C05421=1105.460,240.179,428.078,179.305,14.265,151.128
C05422=1105.455,239.930,428.104,179.301,14.265,151.129
C05423=1105.449,239.682,428.131,179.297,14.266,151.129
C05424=1105.443,239.434,428.158,179.293,14.266,151.130
C05425=1105.437,239.185,428.184,179.289,14.266,151.131
C05426=1105.432,238.936,428.210,179.285,14.266,151.132
C05427=1105.426,238.688,428.237,179.281,14.266,151.133
C05428=1105.420,238.440,428.263,179.277,14.266,151.134
C05429=1105.415,238.191,428.289,179.274,14.266,151.135
C05430=1105.409,237.942,428.316,179.270,14.266,151.136
C05431=1105.404,237.693,428.342,179.266,14.266,151.137
C05432=1105.398,237.445,428.369,179.262,14.267,151.138
C05433=1105.393,237.197,428.395,179.258,14.267,151.139
C05434=1105.387,236.948,428.421,179.254,14.267,151.139
C05435=1105.379,236.586,428.459,179.248,14.266,151.141
C05436=1105.370,236.224,428.498,179.242,14.267,151.142
C05437=1105.363,235.862,428.536,179.237,14.267,151.143
C05438=1105.354,235.500,428.574,179.231,14.268,151.145
C05439=1105.348,235.252,428.600,179.227,14.268,151.146
C05440=1105.342,235.003,428.626,179.223,14.268,151.147
C05441=1105.336,234.754,428.653,179.220,14.268,151.147
C05442=1105.331,234.506,428.678,179.216,14.268,151.148
C05443=1105.326,234.257,428.704,179.211,14.268,151.149
C05444=1105.320,234.009,428.731,179.208,14.268,151.150
C05445=1105.315,233.760,428.757,179.204,14.268,151.151
C05446=1105.308,233.512,428.783,179.200,14.268,151.152
C05447=1105.303,233.263,428.809,179.196,14.269,151.153
C05448=1105.297,233.014,428.835,179.192,14.269,151.154
C05449=1105.292,232.765,428.861,179.188,14.269,151.155
C05450=1105.286,232.516,428.887,179.184,14.269,151.156
C05451=1105.280,232.269,428.913,179.180,14.269,151.157
C05452=1105.275,232.020,428.939,179.176,14.269,151.157
C05453=1105.269,231.771,428.965,179.172,14.270,151.159
C05454=1105.264,231.522,428.991,179.168,14.270,151.159
C05455=1105.257,231.274,429.017,179.164,14.270,151.160
C05456=1105.252,231.025,429.043,179.160,14.270,151.161
C05457=1105.247,230.777,429.068,179.156,14.270,151.162
C05458=1105.241,230.529,429.095,179.152,14.270,151.163
C05459=1105.235,230.280,429.120,179.148,14.270,151.164
C05460=1105.229,230.031,429.146,179.145,14.271,151.165
C05461=1105.224,229.782,429.172,179.141,14.271,151.166
C05462=1105.218,229.533,429.198,179.137,14.272,151.167
C05463=1105.213,229.286,429.224,179.133,14.272,151.168
C05464=1105.206,229.037,429.249,179.129,14.272,151.169
C05465=1105.201,228.788,429.275,179.125,14.272,151.170
C05466=1105.195,228.539,429.301,179.121,14.272,151.171
C05467=1105.189,228.290,429.326,179.117,14.272,151.171
C05468=1105.184,228.041,429.352,179.113,14.272,151.172
C05469=1105.178,227.794,429.378,179.109,14.273,151.173
C05470=1105.172,227.545,429.404,179.105,14.273,151.174
C05471=1105.167,227.296,429.430,179.101,14.273,151.175
C05472=1105.161,227.047,429.455,179.097,14.273,151.176
C05473=1105.156,226.799,429.481,179.094,14.274,151.177
C05474=1105.150,226.550,429.506,179.090,14.274,151.178
C05475=1105.144,226.301,429.532,179.086,14.274,151.179
C05476=1105.138,226.053,429.557,179.082,14.275,151.180
C05477=1105.133,225.804,429.583,179.078,14.275,151.181
C05478=1105.127,225.556,429.608,179.074,14.275,151.182
C05479=1105.121,225.307,429.634,179.070,14.275,151.183
C05480=1105.115,225.058,429.660,179.066,14.276,151.184
C05481=1105.110,224.810,429.685,179.062,14.276,151.185
C05482=1105.104,224.561,429.710,179.058,14.276,151.185
C05483=1105.099,224.312,429.736,179.055,14.276,151.186
C05484=1105.092,224.064,429.762,179.051,14.277,151.187
C05485=1105.088,223.815,429.787,179.047,14.277,151.188
C05486=1105.081,223.567,429.813,179.043,14.277,151.189
C05487=1105.074,223.196,429.851,179.037,14.277,151.191
C05488=1105.065,222.825,429.888,179.031,14.278,151.192
C05489=1105.057,222.456,429.926,179.026,14.278,151.193
C05490=1105.048,222.085,429.964,179.020,14.279,151.195
C05491=1105.042,221.836,429.990,179.016,14.279,151.196
C05492=1105.037,221.588,430.014,179.012,14.279,151.197
C05493=1105.031,221.339,430.040,179.008,14.280,151.198
C05494=1105.025,221.090,430.065,179.004,14.280,151.199
C05495=1105.020,220.842,430.090,179.000,14.280,151.199
C05496=1105.014,220.593,430.116,178.996,14.280,151.201
C05497=1105.008,220.344,430.141,178.992,14.280,151.201
C05498=1105.003,220.096,430.166,178.989,14.281,151.202
C05499=1104.997,219.847,430.191,178.985,14.282,151.203
C05500=1104.991,219.597,430.217,178.981,14.282,151.204
C05501=1104.986,219.349,430.241,178.977,14.282,151.205
C05502=1104.980,219.101,430.267,178.973,14.282,151.206
C05503=1104.973,218.852,430.292,178.969,14.282,151.207
C05504=1104.969,218.603,430.317,178.965,14.283,151.208
C05505=1104.963,218.355,430.342,178.961,14.283,151.209
C05506=1104.957,218.107,430.367,178.957,14.284,151.210
C05507=1104.951,217.857,430.392,178.954,14.284,151.211
C05508=1104.946,217.608,430.418,178.949,14.284,151.212
C05509=1104.940,217.360,430.442,178.945,14.284,151.213
C05510=1104.934,217.111,430.467,178.942,14.285,151.214
C05511=1104.929,216.863,430.492,178.937,14.285,151.215
C05512=1104.923,216.614,430.517,178.933,14.285,151.216
C05513=1104.918,216.366,430.543,178.930,14.286,151.216
C05514=1104.912,216.116,430.567,178.926,14.286,151.218
C05515=1104.906,215.868,430.593,178.922,14.287,151.218
C05516=1104.900,215.619,430.617,178.918,14.287,151.219
C05517=1104.894,215.370,430.642,178.914,14.287,151.220
C05518=1104.890,215.121,430.667,178.910,14.287,151.221
C05519=1104.883,214.873,430.692,178.906,14.287,151.222
C05520=1104.878,214.624,430.717,178.903,14.288,151.223
C05521=1104.872,214.375,430.742,178.899,14.289,151.224
C05522=1104.867,214.127,430.766,178.895,14.289,151.225
C05523=1104.860,213.878,430.792,178.891,14.289,151.226
C05524=1104.856,213.629,430.816,178.887,14.289,151.227
C05525=1104.850,213.380,430.841,178.883,14.289,151.228
C05526=1104.844,213.132,430.866,178.879,14.291,151.229
C05527=1104.839,212.883,430.891,178.876,14.291,151.230
C05528=1104.833,212.635,430.916,178.871,14.291,151.231
C05529=1104.827,212.386,430.940,178.867,14.291,151.232
C05530=1104.822,212.137,430.964,178.864,14.291,151.233
C05531=1104.816,211.888,430.990,178.859,14.292,151.234
C05532=1104.810,211.640,431.014,178.856,14.293,151.235
C05533=1104.804,211.390,431.039,178.852,14.293,151.236
C05534=1104.799,211.142,431.064,178.848,14.293,151.237
C05535=1104.793,210.893,431.088,178.844,14.293,151.237
C05536=1104.787,210.645,431.113,178.840,14.294,151.238
C05537=1104.782,210.396,431.137,178.836,14.294,151.239
C05538=1104.776,210.147,431.162,178.833,14.295,151.240
C05539=1104.768,209.781,431.198,178.826,14.295,151.242
C05540=1104.759,209.413,431.234,178.821,14.296,151.243
C05541=1104.752,209.046,431.270,178.815,14.296,151.245
C05542=1104.743,208.679,431.307,178.810,14.297,151.246
C05543=1104.720,207.682,431.405,178.783,14.296,151.252
C05544=1104.714,207.433,431.429,178.779,14.297,151.253
C05545=1104.709,207.184,431.453,178.774,14.298,151.254
C05546=1104.703,206.936,431.477,178.770,14.299,151.256
C05547=1104.697,206.687,431.502,178.766,14.301,151.257
C05548=1104.691,206.438,431.526,178.761,14.302,151.258
C05549=1104.686,206.190,431.550,178.758,14.303,151.259
C05550=1104.679,205.941,431.574,178.753,14.304,151.260
C05551=1104.674,205.692,431.599,178.749,14.306,151.262
C05552=1104.668,205.443,431.623,178.745,14.307,151.263
C05553=1104.663,205.194,431.647,178.741,14.308,151.264
C05554=1104.657,204.946,431.671,178.737,14.309,151.265
C05555=1104.651,204.697,431.696,178.733,14.311,151.266
C05556=1104.646,204.448,431.720,178.728,14.312,151.268
C05557=1104.640,204.200,431.744,178.724,14.312,151.269
C05558=1104.634,203.951,431.768,178.720,14.314,151.270
C05559=1104.628,203.702,431.793,178.716,14.315,151.271
C05560=1104.623,203.453,431.817,178.712,14.316,151.272
C05561=1104.617,203.205,431.840,178.708,14.317,151.273
C05562=1104.611,202.956,431.865,178.704,14.319,151.275
C05563=1104.606,202.707,431.889,178.699,14.319,151.276
C05564=1104.600,202.458,431.912,178.695,14.321,151.277
C05565=1104.594,202.209,431.937,178.691,14.322,151.278
C05566=1104.588,201.961,431.961,178.687,14.323,151.279
C05567=1104.583,201.712,431.985,178.683,14.324,151.281
C05568=1104.577,201.463,432.009,178.678,14.325,151.282
C05569=1104.571,201.215,432.033,178.674,14.327,151.283
C05570=1104.566,200.965,432.057,178.670,14.327,151.284
C05571=1104.559,200.716,432.081,178.666,14.329,151.285
C05572=1104.554,200.468,432.105,178.662,14.330,151.287
C05573=1104.548,200.220,432.129,178.658,14.331,151.288
C05574=1104.542,199.970,432.153,178.654,14.332,151.289
C05575=1104.536,199.721,432.176,178.650,14.334,151.290
C05576=1104.531,199.473,432.200,178.645,14.335,151.291
C05577=1104.525,199.225,432.224,178.642,14.336,151.292
C05578=1104.520,198.975,432.248,178.637,14.337,151.294
C05579=1104.513,198.726,432.272,178.633,14.339,151.295
C05580=1104.508,198.478,432.296,178.629,14.339,151.296
C05581=1104.502,198.229,432.320,178.625,14.341,151.297
C05582=1104.496,197.980,432.343,178.621,14.342,151.298
C05583=1104.491,197.731,432.367,178.617,14.343,151.299
C05584=1104.485,197.482,432.390,178.613,14.344,151.301
C05585=1104.479,197.234,432.414,178.609,14.345,151.302
C05586=1104.473,196.985,432.438,178.605,14.347,151.303
C05587=1104.468,196.736,432.462,178.600,14.348,151.304
C05588=1104.462,196.487,432.486,178.597,14.349,151.305
C05589=1104.457,196.238,432.509,178.592,14.350,151.307
C05590=1104.451,195.990,432.533,178.589,14.351,151.308
C05591=1104.444,195.741,432.557,178.584,14.352,151.309
C05592=1104.439,195.492,432.580,178.581,14.353,151.310
C05593=1104.433,195.243,432.604,178.576,14.354,151.311
C05594=1104.428,194.994,432.627,178.572,14.356,151.312
C05595=1104.422,194.746,432.651,178.568,14.356,151.313
C05596=1104.416,194.497,432.674,178.564,14.358,151.315
C05597=1104.410,194.248,432.699,178.560,14.359,151.316
C05598=1104.405,193.999,432.722,178.555,14.360,151.317
C05599=1104.399,193.751,432.745,178.552,14.361,151.318
C05600=1104.394,193.501,432.769,178.547,14.362,151.319
C05601=1104.388,193.252,432.792,178.544,14.363,151.320
C05602=1104.382,193.004,432.815,178.540,14.364,151.321
C05603=1104.377,192.755,432.839,178.536,14.365,151.323
C05604=1104.370,192.483,432.865,178.531,14.366,151.324
C05605=1104.364,192.212,432.890,178.527,14.367,151.325
C05606=1104.358,191.941,432.916,178.523,14.369,151.326
C05607=1104.352,191.670,432.941,178.518,14.370,151.328
C05608=1104.346,191.421,432.964,178.514,14.371,151.329
C05609=1104.341,191.172,432.989,178.510,14.372,151.330
C05610=1104.335,190.923,433.012,178.506,14.373,151.331
C05611=1104.329,190.674,433.034,178.502,14.375,151.332
C05612=1104.323,190.425,433.059,178.498,14.375,151.333
C05613=1104.318,190.176,433.082,178.494,14.377,151.334
C05614=1104.312,189.927,433.105,178.490,14.378,151.336
C05615=1104.306,189.678,433.128,178.486,14.379,151.337
C05616=1104.301,189.430,433.152,178.482,14.379,151.338
C05617=1104.295,189.181,433.175,178.478,14.380,151.339
C05618=1104.290,188.932,433.198,178.474,14.382,151.340
C05619=1104.284,188.683,433.221,178.470,14.382,151.341
C05620=1104.278,188.435,433.245,178.466,14.384,151.342
C05621=1104.273,188.186,433.268,178.462,14.385,151.343
C05622=1104.267,187.937,433.291,178.458,14.386,151.345
C05623=1104.261,187.688,433.314,178.454,14.386,151.346
C05624=1104.256,187.439,433.338,178.450,14.388,151.347
C05625=1104.251,187.190,433.361,178.446,14.389,151.348
C05626=1104.245,186.941,433.384,178.442,14.390,151.349
C05627=1104.239,186.693,433.407,178.438,14.391,151.350
C05628=1104.233,186.444,433.430,178.434,14.392,151.351
C05629=1104.228,186.195,433.454,178.430,14.393,151.352
C05630=1104.222,185.946,433.477,178.426,14.393,151.353
C05631=1104.217,185.697,433.499,178.422,14.395,151.354
C05632=1104.211,185.449,433.522,178.418,14.396,151.356
C05633=1104.206,185.200,433.545,178.414,14.397,151.357
C05634=1104.200,184.951,433.568,178.410,14.398,151.358
C05635=1104.194,184.702,433.591,178.407,14.399,151.359
C05636=1104.189,184.453,433.614,178.402,14.400,151.360
C05637=1104.183,184.204,433.637,178.399,14.401,151.361
C05638=1104.176,183.954,433.660,178.394,14.402,151.362
C05639=1104.171,183.706,433.683,178.391,14.403,151.364
C05640=1104.165,183.457,433.706,178.386,14.404,151.365
C05641=1104.159,183.208,433.729,178.383,14.405,151.366
C05642=1104.154,182.959,433.752,178.378,14.406,151.367
C05643=1104.148,182.710,433.775,178.375,14.408,151.368
C05644=1104.141,182.461,433.797,178.371,14.408,151.369
C05645=1104.136,182.212,433.820,178.367,14.410,151.370
C05646=1104.130,181.964,433.843,178.363,14.411,151.371
C05647=1104.125,181.715,433.866,178.359,14.412,151.372
C05648=1104.119,181.466,433.889,178.355,14.412,151.374
C05649=1104.113,181.218,433.912,178.351,14.414,151.375
C05650=1104.108,180.969,433.935,178.347,14.415,151.376
C05651=1104.101,180.720,433.957,178.343,14.416,151.377
C05652=1104.096,180.471,433.979,178.339,14.417,151.378
C05653=1104.090,180.222,434.002,178.336,14.418,151.379
C05654=1104.084,179.973,434.025,178.331,14.419,151.380
C05655=1104.078,179.724,434.048,178.328,14.420,151.381
C05656=1104.073,179.475,434.071,178.323,14.421,151.382
C05657=1104.067,179.226,434.093,178.320,14.422,151.383
C05658=1104.061,178.977,434.116,178.316,14.423,151.385
C05659=1104.055,178.728,434.139,178.312,14.424,151.386
C05660=1104.049,178.479,434.161,178.308,14.425,151.387
C05661=1104.044,178.231,434.184,178.304,14.426,151.388
C05662=1104.038,177.982,434.206,178.300,14.427,151.389
C05663=1104.032,177.733,434.229,178.297,14.428,151.390
C05664=1104.027,177.484,434.252,178.292,14.429,151.391
C05665=1104.021,177.234,434.274,178.288,14.430,151.392
C05666=1104.015,176.985,434.297,178.284,14.431,151.393
C05667=1104.009,176.737,434.319,178.280,14.432,151.394
C05668=1104.003,176.465,434.344,178.277,14.433,151.395
C05669=1103.997,176.194,434.368,178.272,14.434,151.397
C05670=1103.991,175.922,434.393,178.268,14.435,151.398
C05671=1103.985,175.650,434.418,178.263,14.436,151.399
C05672=1103.979,175.401,434.439,178.260,14.437,151.400
C05673=1103.973,175.152,434.462,178.255,14.438,151.401
C05674=1103.967,174.903,434.485,178.252,14.439,151.402
C05675=1103.961,174.654,434.507,178.248,14.439,151.403
C05676=1103.956,174.406,434.529,178.244,14.441,151.404
C05677=1103.951,174.156,434.552,178.240,14.441,151.405
C05678=1103.945,173.907,434.575,178.237,14.443,151.407
C05679=1103.939,173.658,434.596,178.232,14.443,151.408
C05680=1103.934,173.410,434.619,178.229,14.445,151.409
C05681=1103.928,173.160,434.641,178.225,14.445,151.410
C05682=1103.922,172.912,434.663,178.221,14.447,151.411
C05683=1103.916,172.662,434.686,178.217,14.447,151.412
C05684=1103.911,172.414,434.708,178.214,14.448,151.413
C05685=1103.905,172.165,434.730,178.209,14.449,151.414
C05686=1103.899,171.916,434.753,178.206,14.450,151.415
C05687=1103.894,171.667,434.775,178.202,14.451,151.416
C05688=1103.888,171.419,434.797,178.198,14.452,151.417
C05689=1103.883,171.169,434.819,178.194,14.453,151.418
C05690=1103.877,170.920,434.842,178.191,14.453,151.419
C05691=1103.871,170.671,434.864,178.187,14.454,151.420
C05692=1103.866,170.422,434.886,178.183,14.455,151.421
C05693=1103.859,170.174,434.908,178.179,14.456,151.422
C05694=1103.854,169.924,434.930,178.175,14.457,151.423
C05695=1103.849,169.675,434.952,178.172,14.458,151.424
C05696=1103.843,169.427,434.974,178.168,14.459,151.425
C05697=1103.837,169.177,434.997,178.164,14.459,151.426
C05698=1103.832,168.929,435.018,178.160,14.461,151.427
C05699=1103.826,168.680,435.041,178.156,14.461,151.428
C05700=1103.821,168.430,435.063,178.153,14.462,151.429
C05701=1103.815,168.182,435.084,178.149,14.463,151.431
C05702=1103.809,167.933,435.107,178.145,14.464,151.432
C05703=1103.803,167.684,435.129,178.141,14.464,151.432
C05704=1103.798,167.435,435.151,178.138,14.466,151.434
C05705=1103.792,167.186,435.172,178.134,14.466,151.435
C05706=1103.786,166.937,435.195,178.130,14.467,151.436
C05707=1103.782,166.688,435.217,178.126,14.468,151.437
C05708=1103.775,166.439,435.239,178.123,14.469,151.438
C05709=1103.771,166.190,435.261,178.119,14.470,151.439
C05710=1103.764,165.941,435.282,178.115,14.470,151.440
C05711=1103.759,165.692,435.305,178.111,14.471,151.441
C05712=1103.753,165.443,435.327,178.107,14.472,151.442
C05713=1103.748,165.194,435.349,178.104,14.473,151.443
C05714=1103.742,164.945,435.370,178.100,14.473,151.444
C05715=1103.737,164.696,435.392,178.096,14.475,151.445
C05716=1103.731,164.447,435.414,178.092,14.475,151.446
C05717=1103.726,164.198,435.436,178.089,14.476,151.447
C05718=1103.719,163.949,435.458,178.085,14.477,151.448
C05719=1103.714,163.700,435.480,178.081,14.478,151.449
C05720=1103.708,163.451,435.502,178.077,14.478,151.450
C05721=1103.703,163.202,435.524,178.074,14.479,151.451
C05722=1103.697,162.953,435.545,178.070,14.480,151.452
C05723=1103.692,162.704,435.567,178.067,14.481,151.453
C05724=1103.686,162.455,435.589,178.062,14.481,151.454
C05725=1103.681,162.207,435.610,178.059,14.482,151.455
C05726=1103.675,161.957,435.632,178.055,14.483,151.456
C05727=1103.670,161.709,435.653,178.052,14.484,151.457
C05728=1103.664,161.459,435.676,178.048,14.485,151.458
C05729=1103.659,161.211,435.697,178.045,14.485,151.459
C05730=1103.653,160.961,435.719,178.040,14.486,151.460
C05731=1103.647,160.713,435.740,178.037,14.487,151.461
C05732=1103.641,160.440,435.764,178.033,14.488,151.462
C05733=1103.634,160.168,435.788,178.028,14.489,151.463
C05734=1103.628,159.896,435.811,178.025,14.490,151.464
C05735=1103.622,159.624,435.835,178.021,14.491,151.465
C05736=1103.617,159.375,435.856,178.017,14.491,151.466
C05737=1103.610,159.126,435.878,178.013,14.492,151.467
C05738=1103.605,158.877,435.899,178.009,14.493,151.468
C05739=1103.599,158.628,435.921,178.006,14.494,151.469
C05740=1103.594,158.379,435.942,178.002,14.494,151.470
C05741=1103.588,158.130,435.963,177.998,14.495,151.471
C05742=1103.582,157.881,435.985,177.995,14.496,151.472
C05743=1103.576,157.632,436.006,177.991,14.497,151.473
C05744=1103.571,157.383,436.028,177.987,14.497,151.474
C05745=1103.565,157.134,436.050,177.984,14.498,151.475
C05746=1103.560,156.885,436.070,177.980,14.499,151.476
C05747=1103.554,156.635,436.092,177.977,14.500,151.477
C05748=1103.548,156.387,436.113,177.972,14.500,151.478
C05749=1103.542,156.138,436.135,177.969,14.501,151.479
C05750=1103.538,155.888,436.156,177.965,14.502,151.480
C05751=1103.531,155.639,436.178,177.962,14.503,151.481
C05752=1103.526,155.391,436.199,177.958,14.503,151.482
C05753=1103.520,155.142,436.220,177.955,14.504,151.483
C05754=1103.515,154.892,436.241,177.950,14.505,151.484
C05755=1103.509,154.644,436.262,177.947,14.506,151.485
C05756=1103.503,154.395,436.284,177.943,14.506,151.485
C05757=1103.498,154.145,436.305,177.940,14.507,151.487
C05758=1103.491,153.896,436.326,177.936,14.508,151.487
C05759=1103.486,153.648,436.347,177.933,14.508,151.488
C05760=1103.480,153.398,436.368,177.929,14.509,151.489
C05761=1103.474,153.149,436.390,177.925,14.510,151.490
C05762=1103.469,152.901,436.411,177.922,14.510,151.491
C05763=1103.463,152.651,436.432,177.918,14.512,151.492
C05764=1103.457,152.403,436.453,177.914,14.512,151.493
C05765=1103.451,152.153,436.475,177.911,14.513,151.494
C05766=1103.447,151.904,436.496,177.907,14.513,151.495
C05767=1103.441,151.655,436.517,177.904,14.514,151.496
C05768=1103.435,151.406,436.538,177.900,14.515,151.497
C05769=1103.430,151.157,436.559,177.897,14.516,151.498
C05770=1103.423,150.908,436.580,177.893,14.516,151.499
C05771=1103.418,150.659,436.601,177.889,14.517,151.500
C05772=1103.412,150.410,436.621,177.886,14.518,151.501
C05773=1103.406,150.161,436.643,177.882,14.518,151.502
C05774=1103.401,149.912,436.664,177.879,14.519,151.503
C05775=1103.395,149.663,436.685,177.875,14.519,151.504
C05776=1103.390,149.413,436.706,177.872,14.521,151.505
C05777=1103.384,149.165,436.727,177.868,14.521,151.506
C05778=1103.379,148.916,436.748,177.864,14.522,151.506
C05779=1103.373,148.666,436.769,177.861,14.522,151.507
C05780=1103.367,148.417,436.790,177.857,14.523,151.508
C05781=1103.362,148.169,436.811,177.853,14.523,151.509
C05782=1103.356,147.919,436.832,177.850,14.524,151.510
C05783=1103.350,147.670,436.852,177.846,14.525,151.511
C05784=1103.344,147.422,436.873,177.843,14.526,151.512
C05785=1103.338,147.172,436.894,177.839,14.526,151.513
C05786=1103.333,146.923,436.915,177.836,14.527,151.514
C05787=1103.328,146.674,436.936,177.832,14.527,151.515
C05788=1103.322,146.424,436.957,177.829,14.528,151.516
C05789=1103.315,146.176,436.978,177.825,14.529,151.517
C05790=1103.310,145.927,436.998,177.822,14.530,151.518
C05791=1103.304,145.677,437.019,177.817,14.530,151.519
C05792=1103.299,145.429,437.040,177.814,14.531,151.520
C05793=1103.293,145.180,437.060,177.810,14.531,151.520
C05794=1103.287,144.930,437.081,177.807,14.532,151.521
C05795=1103.281,144.682,437.103,177.803,14.533,151.522
C05796=1103.275,144.409,437.125,177.800,14.534,151.523
C05797=1103.269,144.136,437.148,177.796,14.534,151.524
C05798=1103.264,143.864,437.170,177.792,14.535,151.525
C05799=1103.257,143.592,437.192,177.788,14.535,151.526
C05800=1103.251,143.342,437.213,177.785,14.536,151.527
C05801=1103.245,143.094,437.234,177.781,14.537,151.528
C05802=1103.240,142.845,437.255,177.778,14.537,151.529
C05803=1103.234,142.596,437.275,177.774,14.538,151.530
C05804=1103.228,142.346,437.296,177.770,14.539,151.531
C05805=1103.223,142.097,437.316,177.768,14.539,151.532
C05806=1103.217,141.848,437.337,177.764,14.539,151.532
C05807=1103.211,141.600,437.357,177.761,14.540,151.533
C05808=1103.206,141.351,437.378,177.757,14.541,151.534
C05809=1103.200,141.101,437.399,177.754,14.541,151.535
C05810=1103.194,140.852,437.419,177.750,14.542,151.536
C05811=1103.189,140.603,437.439,177.746,14.543,151.537
C05812=1103.184,140.354,437.460,177.743,14.543,151.538
C05813=1103.178,140.105,437.480,177.739,14.544,151.539
C05814=1103.172,139.855,437.501,177.735,14.544,151.540
C05815=1103.166,139.606,437.521,177.733,14.545,151.541
C05816=1103.160,139.358,437.542,177.729,14.545,151.541
C05817=1103.155,139.109,437.563,177.726,14.546,151.542
C05818=1103.149,138.860,437.583,177.722,14.546,151.543
C05819=1103.144,138.611,437.603,177.719,14.547,151.544
C05820=1103.137,138.361,437.623,177.715,14.547,151.545
C05821=1103.132,138.112,437.644,177.711,14.548,151.546
C05822=1103.127,137.863,437.665,177.708,14.548,151.547
C05823=1103.121,137.614,437.685,177.705,14.549,151.548
C05824=1103.116,137.365,437.705,177.702,14.550,151.549
C05825=1103.110,137.116,437.725,177.698,14.550,151.549
C05826=1103.104,136.866,437.745,177.694,14.551,151.550
C05827=1103.098,136.617,437.765,177.691,14.551,151.551
C05828=1103.093,136.368,437.786,177.688,14.552,151.552
C05829=1103.087,136.119,437.806,177.684,14.552,151.553
C05830=1103.081,135.870,437.826,177.681,14.553,151.554
C05831=1103.075,135.621,437.846,177.677,14.553,151.555
C05832=1103.070,135.372,437.867,177.674,14.554,151.556
C05833=1103.064,135.122,437.887,177.670,14.554,151.556
C05834=1103.058,134.873,437.908,177.667,14.555,151.557
C05835=1103.052,134.624,437.928,177.663,14.555,151.558
C05836=1103.047,134.375,437.947,177.660,14.556,151.559
C05837=1103.041,134.126,437.967,177.656,14.556,151.560
C05838=1103.035,133.877,437.987,177.653,14.557,151.561
C05839=1103.030,133.628,438.008,177.649,14.557,151.562
C05840=1103.024,133.379,438.028,177.646,14.558,151.562
C05841=1103.019,133.129,438.048,177.643,14.558,151.563
C05842=1103.013,132.881,438.068,177.640,14.559,151.564
C05843=1103.008,132.631,438.088,177.636,14.560,151.565
C05844=1103.002,132.383,438.108,177.633,14.560,151.566
C05845=1102.996,132.134,438.128,177.630,14.561,151.567
C05846=1102.990,131.883,438.148,177.626,14.561,151.568
C05847=1102.984,131.635,438.168,177.623,14.561,151.568
C05848=1102.978,131.386,438.188,177.619,14.562,151.569
C05849=1102.973,131.137,438.209,177.616,14.563,151.570
C05850=1102.968,130.887,438.228,177.612,14.562,151.571
C05851=1102.962,130.638,438.248,177.609,14.563,151.572
C05852=1102.956,130.390,438.268,177.605,14.564,151.573
C05853=1102.951,130.140,438.288,177.602,14.564,151.574
C05854=1102.945,129.891,438.308,177.598,14.565,151.574
C05855=1102.939,129.642,438.328,177.596,14.565,151.575
C05856=1102.933,129.393,438.347,177.592,14.566,151.576
C05857=1102.928,129.144,438.368,177.589,14.566,151.577
C05858=1102.921,128.894,438.388,177.586,14.567,151.578
C05859=1102.915,128.645,438.407,177.582,14.567,151.579
C05860=1102.909,128.373,438.429,177.578,14.567,151.580
C05861=1102.903,128.100,438.451,177.575,14.568,151.580
C05862=1102.897,127.827,438.472,177.571,14.569,151.581
C05863=1102.890,127.555,438.494,177.567,14.569,151.582
C05864=1102.885,127.306,438.513,177.564,14.569,151.583
C05865=1102.880,127.057,438.533,177.560,14.570,151.584
C05866=1102.874,126.807,438.553,177.557,14.570,151.585
C05867=1102.868,126.558,438.573,177.554,14.571,151.586
C05868=1102.862,126.310,438.593,177.551,14.571,151.586
C05869=1102.856,126.060,438.612,177.548,14.572,151.587
C05870=1102.850,125.811,438.632,177.544,14.572,151.588
C05871=1102.845,125.562,438.652,177.541,14.572,151.589
C05872=1102.839,125.313,438.672,177.537,14.573,151.590
C05873=1102.834,125.063,438.691,177.534,14.573,151.590
C05874=1102.828,124.814,438.710,177.530,14.574,151.591
C05875=1102.822,124.565,438.730,177.527,14.574,151.592
C05876=1102.816,124.316,438.749,177.524,14.574,151.593
C05877=1102.810,124.067,438.769,177.521,14.575,151.594
C05878=1102.805,123.817,438.789,177.518,14.575,151.595
C05879=1102.799,123.568,438.809,177.514,14.575,151.595
C05880=1102.794,123.319,438.828,177.511,14.576,151.596
C05881=1102.788,123.070,438.847,177.508,14.576,151.597
C05882=1102.782,122.821,438.867,177.504,14.577,151.598
C05883=1102.777,122.572,438.886,177.501,14.577,151.599
C05884=1102.771,122.323,438.906,177.498,14.577,151.599
C05885=1102.765,122.074,438.926,177.494,14.577,151.600
C05886=1102.759,121.824,438.945,177.491,14.578,151.601
C05887=1102.754,121.575,438.965,177.488,14.578,151.602
C05888=1102.748,121.326,438.985,177.485,14.579,151.603
C05889=1102.743,121.076,439.004,177.481,14.579,151.603
C05890=1102.738,120.828,439.023,177.478,14.580,151.604
C05891=1102.732,120.579,439.043,177.475,14.580,151.605
C05892=1102.726,120.329,439.062,177.472,14.580,151.606
C05893=1102.720,120.080,439.081,177.469,14.581,151.607
C05894=1102.715,119.830,439.100,177.465,14.581,151.607
C05895=1102.709,119.582,439.120,177.462,14.581,151.608
C05896=1102.704,119.333,439.139,177.459,14.581,151.609
C05897=1102.698,119.083,439.158,177.456,14.582,151.610
C05898=1102.692,118.834,439.178,177.452,14.582,151.611
C05899=1102.686,118.585,439.197,177.449,14.582,151.611
C05900=1102.680,118.336,439.217,177.445,14.582,151.612
C05901=1102.675,118.086,439.236,177.443,14.583,151.613
C05902=1102.670,117.838,439.255,177.440,14.583,151.613
C05903=1102.664,117.588,439.274,177.436,14.583,151.614
C05904=1102.658,117.339,439.294,177.433,14.584,151.615
C05905=1102.653,117.089,439.313,177.430,14.584,151.616
C05906=1102.648,116.841,439.332,177.427,14.585,151.617
C05907=1102.642,116.592,439.352,177.423,14.585,151.617
C05908=1102.636,116.342,439.371,177.420,14.585,151.618
C05909=1102.630,116.093,439.390,177.416,14.585,151.619
C05910=1102.625,115.844,439.409,177.414,14.585,151.620
C05911=1102.619,115.595,439.428,177.410,14.585,151.620
C05912=1102.614,115.345,439.447,177.407,14.586,151.621
C05913=1102.608,115.096,439.467,177.404,14.586,151.622
C05914=1102.603,114.847,439.486,177.401,14.586,151.623
C05915=1102.597,114.598,439.505,177.398,14.587,151.623
C05916=1102.592,114.348,439.524,177.394,14.587,151.624
C05917=1102.586,114.099,439.543,177.392,14.587,151.625
C05918=1102.580,113.850,439.562,177.388,14.587,151.626
C05919=1102.574,113.601,439.581,177.385,14.588,151.626
C05920=1102.569,113.352,439.600,177.382,14.588,151.627
C05921=1102.563,113.102,439.619,177.379,14.588,151.628
C05922=1102.558,112.853,439.638,177.376,14.589,151.629
C05923=1102.551,112.604,439.657,177.372,14.588,151.629
C05924=1102.545,112.331,439.678,177.368,14.589,151.630
C05925=1102.539,112.059,439.699,177.366,14.589,151.631
C05926=1102.533,111.786,439.719,177.362,14.589,151.632
C05927=1102.527,111.513,439.741,177.358,14.590,151.633
C05928=1102.521,111.265,439.759,177.355,14.590,151.634
C05929=1102.515,111.016,439.778,177.352,14.591,151.634
C05930=1102.510,110.766,439.797,177.349,14.590,151.635
C05931=1102.504,110.517,439.816,177.346,14.591,151.636
C05932=1102.498,110.268,439.834,177.342,14.591,151.637
C05933=1102.493,110.018,439.853,177.340,14.591,151.637
C05934=1102.487,109.769,439.873,177.336,14.591,151.638
C05935=1102.481,109.520,439.891,177.333,14.592,151.639
C05936=1102.475,109.271,439.910,177.330,14.592,151.640
C05937=1102.470,109.021,439.929,177.327,14.592,151.640
C05938=1102.464,108.772,439.947,177.324,14.592,151.641
C05939=1102.459,108.523,439.966,177.321,14.592,151.642
C05940=1102.453,108.274,439.986,177.318,14.593,151.642
C05941=1102.446,108.024,440.004,177.314,14.593,151.643
C05942=1102.441,107.776,440.023,177.311,14.593,151.644
C05943=1102.435,107.526,440.041,177.308,14.593,151.645
C05944=1102.430,107.277,440.060,177.305,14.594,151.645
C05945=1102.424,107.028,440.079,177.302,14.594,151.646
C05946=1102.418,106.779,440.098,177.299,14.594,151.647
C05947=1102.413,106.529,440.116,177.296,14.594,151.647
C05948=1102.408,106.280,440.135,177.292,14.594,151.648
C05949=1102.401,106.031,440.154,177.290,14.595,151.649
C05950=1102.396,105.781,440.172,177.286,14.594,151.650
C05951=1102.390,105.532,440.191,177.283,14.595,151.650
C05952=1102.384,105.283,440.210,177.281,14.595,151.651
C05953=1102.379,105.034,440.228,177.277,14.595,151.652
C05954=1102.373,104.784,440.247,177.274,14.596,151.653
C05955=1102.368,104.536,440.266,177.271,14.595,151.653
C05956=1102.362,104.286,440.283,177.268,14.596,151.654
C05957=1102.356,104.036,440.303,177.264,14.595,151.655
C05958=1102.350,103.788,440.321,177.262,14.596,151.655
C05959=1102.345,103.538,440.340,177.259,14.596,151.656
C05960=1102.339,103.290,440.358,177.256,14.596,151.657
C05961=1102.334,103.040,440.376,177.253,14.597,151.657
C05962=1102.328,102.790,440.396,177.249,14.596,151.658
C05963=1102.322,102.542,440.414,177.247,14.596,151.659
C05964=1102.317,102.292,440.432,177.243,14.596,151.660
C05965=1102.311,102.043,440.451,177.241,14.596,151.660
C05966=1102.306,101.793,440.469,177.238,14.597,151.661
C05967=1102.300,101.545,440.487,177.234,14.597,151.662
C05968=1102.294,101.295,440.506,177.232,14.597,151.662
C05969=1102.289,101.046,440.524,177.228,14.597,151.663
C05970=1102.283,100.796,440.543,177.225,14.597,151.664
C05971=1102.277,100.547,440.561,177.222,14.597,151.664
C05972=1102.271,100.298,440.579,177.219,14.597,151.665
C05973=1102.266,100.049,440.598,177.216,14.598,151.666
C05974=1102.260,99.800,440.616,177.213,14.597,151.666
C05975=1102.254,99.550,440.634,177.210,14.598,151.667
C05976=1102.249,99.301,440.653,177.207,14.598,151.668
C05977=1102.243,99.051,440.671,177.204,14.598,151.668
C05978=1102.238,98.803,440.689,177.200,14.598,151.669
C05979=1102.232,98.553,440.707,177.198,14.598,151.670
C05980=1102.225,98.304,440.726,177.195,14.599,151.671
C05981=1102.220,98.054,440.744,177.191,14.598,151.671
C05982=1102.214,97.805,440.763,177.189,14.599,151.672
C05983=1102.208,97.556,440.780,177.185,14.598,151.673
C05984=1102.203,97.306,440.799,177.183,14.599,151.673
C05985=1102.197,97.058,440.817,177.180,14.599,151.674
C05986=1102.191,96.808,440.835,177.176,14.599,151.675
C05987=1102.186,96.559,440.853,177.174,14.599,151.675
C05988=1102.180,96.286,440.873,177.170,14.599,151.676
C05989=1102.173,96.014,440.893,177.167,14.599,151.677
C05990=1102.167,95.742,440.913,177.164,14.599,151.678
C05991=1102.161,95.469,440.933,177.161,14.599,151.678
C05992=1102.156,95.220,440.951,177.158,14.600,151.679
C05993=1102.150,94.970,440.969,177.155,14.599,151.680
C05994=1102.144,94.722,440.987,177.152,14.600,151.680
C05995=1102.138,94.472,441.005,177.149,14.600,151.681
C05996=1102.133,94.223,441.023,177.146,14.600,151.682
C05997=1102.127,93.973,441.041,177.143,14.600,151.682
C05998=1102.122,93.723,441.059,177.139,14.600,151.683
C05999=1102.115,93.474,441.078,177.137,14.600,151.684
C06000=1102.110,93.225,441.095,177.134,14.599,151.684
C06001=1102.104,92.976,441.113,177.131,14.600,151.685
C06002=1102.099,92.726,441.131,177.128,14.600,151.685
C06003=1102.094,92.477,441.149,177.125,14.600,151.686
C06004=1102.087,92.228,441.168,177.122,14.600,151.687
C06005=1102.082,91.979,441.185,177.119,14.599,151.687
C06006=1102.076,91.730,441.203,177.116,14.600,151.688
C06007=1102.071,91.480,441.221,177.114,14.600,151.689
C06008=1102.065,91.231,441.239,177.110,14.599,151.689
C06009=1102.060,90.982,441.256,177.108,14.600,151.690
C06010=1102.054,90.732,441.274,177.104,14.599,151.691
C06011=1102.048,90.484,441.293,177.102,14.599,151.691
C06012=1102.042,90.234,441.311,177.099,14.600,151.692
C06013=1102.036,89.985,441.328,177.096,14.599,151.693
C06014=1102.031,89.735,441.347,177.093,14.600,151.693
C06015=1102.025,89.486,441.364,177.090,14.600,151.694
C06016=1102.020,89.237,441.382,177.087,14.600,151.695
C06017=1102.014,88.987,441.400,177.084,14.600,151.695
C06018=1102.008,88.738,441.417,177.081,14.600,151.696
C06019=1102.002,88.488,441.435,177.078,14.600,151.696
C06020=1101.996,88.239,441.453,177.075,14.600,151.697
C06021=1101.991,87.990,441.470,177.072,14.600,151.698
C06022=1101.985,87.740,441.488,177.070,14.600,151.698
C06023=1101.979,87.491,441.506,177.066,14.600,151.699
C06024=1101.974,87.242,441.523,177.064,14.600,151.700
C06025=1101.968,86.993,441.541,177.060,14.599,151.700
C06026=1101.962,86.744,441.559,177.058,14.599,151.701
C06027=1101.957,86.495,441.577,177.055,14.600,151.702
C06028=1101.950,86.245,441.594,177.052,14.600,151.702
C06029=1101.945,85.996,441.612,177.049,14.600,151.703
C06030=1101.939,85.747,441.630,177.046,14.599,151.703
C06031=1101.933,85.497,441.648,177.044,14.599,151.704
C06032=1101.928,85.248,441.665,177.041,14.600,151.705
C06033=1101.922,84.999,441.683,177.037,14.599,151.705
C06034=1101.916,84.749,441.700,177.035,14.599,151.706
C06035=1101.911,84.500,441.717,177.032,14.599,151.707
C06036=1101.905,84.250,441.735,177.029,14.599,151.707
C06037=1101.899,84.001,441.753,177.026,14.599,151.708
C06038=1101.894,83.752,441.770,177.023,14.599,151.708
C06039=1101.888,83.503,441.788,177.021,14.599,151.709
C06040=1101.883,83.254,441.806,177.018,14.599,151.710
C06041=1101.877,83.003,441.823,177.015,14.599,151.710
C06042=1101.871,82.754,441.840,177.012,14.599,151.711
C06043=1101.866,82.505,441.858,177.009,14.598,151.711
C06044=1101.860,82.256,441.875,177.006,14.598,151.712
C06045=1101.853,82.007,441.893,177.004,14.599,151.713
C06046=1101.848,81.757,441.910,177.000,14.598,151.713
C06047=1101.843,81.508,441.927,176.998,14.598,151.714
C06048=1101.837,81.259,441.945,176.995,14.598,151.715
C06049=1101.831,81.009,441.963,176.992,14.598,151.715
C06050=1101.826,80.760,441.980,176.990,14.598,151.716
C06051=1101.820,80.511,441.997,176.986,14.598,151.716
C06052=1101.814,80.238,442.017,176.984,14.598,151.717
C06053=1101.808,79.966,442.035,176.980,14.598,151.718
C06054=1101.801,79.693,442.054,176.977,14.597,151.718
C06055=1101.796,79.421,442.073,176.974,14.597,151.719
C06056=1101.790,79.171,442.091,176.971,14.597,151.719
C06057=1101.785,78.921,442.108,176.969,14.597,151.720
C06058=1101.778,78.673,442.125,176.966,14.597,151.721
C06059=1101.773,78.424,442.142,176.963,14.596,151.721
C06060=1101.767,78.173,442.160,176.960,14.597,151.722
C06061=1101.761,77.924,442.177,176.958,14.597,151.722
C06062=1101.756,77.675,442.195,176.955,14.596,151.723
C06063=1101.750,77.426,442.211,176.952,14.596,151.724
C06064=1101.744,77.177,442.228,176.949,14.596,151.724
C06065=1101.738,76.927,442.246,176.946,14.596,151.725
C06066=1101.733,76.677,442.263,176.944,14.596,151.725
C06067=1101.727,76.429,442.280,176.940,14.595,151.726
C06068=1101.722,76.179,442.297,176.938,14.596,151.726
C06069=1101.716,75.930,442.315,176.935,14.596,151.727
C06070=1101.710,75.681,442.331,176.932,14.595,151.728
C06071=1101.704,75.431,442.349,176.930,14.595,151.728
C06072=1101.699,75.181,442.366,176.926,14.595,151.729
C06073=1101.693,74.933,442.383,176.924,14.595,151.729
C06074=1101.687,74.684,442.400,176.921,14.595,151.730
C06075=1101.682,74.434,442.417,176.918,14.595,151.731
C06076=1101.676,74.185,442.435,176.916,14.595,151.731
C06077=1101.670,73.935,442.451,176.913,14.594,151.732
C06078=1101.664,73.686,442.469,176.910,14.594,151.732
C06079=1101.659,73.436,442.486,176.908,14.594,151.733
C06080=1101.653,73.187,442.502,176.904,14.593,151.733
C06081=1101.648,72.938,442.520,176.902,14.593,151.734
C06082=1101.642,72.688,442.536,176.899,14.594,151.735
C06083=1101.636,72.439,442.553,176.896,14.593,151.735
C06084=1101.631,72.190,442.570,176.894,14.593,151.736
C06085=1101.624,71.940,442.588,176.891,14.593,151.736
C06086=1101.619,71.691,442.604,176.888,14.592,151.737
C06087=1101.614,71.441,442.621,176.886,14.592,151.737
C06088=1101.607,71.192,442.638,176.883,14.593,151.738
C06089=1101.602,70.943,442.655,176.880,14.592,151.739
C06090=1101.596,70.694,442.672,176.878,14.592,151.739
C06091=1101.591,70.444,442.689,176.874,14.591,151.740
C06092=1101.585,70.194,442.706,176.872,14.591,151.740
C06093=1101.579,69.946,442.723,176.869,14.591,151.741
C06094=1101.574,69.696,442.740,176.866,14.591,151.741
C06095=1101.568,69.447,442.756,176.864,14.591,151.742
C06096=1101.562,69.197,442.774,176.861,14.591,151.742
C06097=1101.556,68.948,442.790,176.858,14.590,151.743
C06098=1101.551,68.698,442.807,176.855,14.590,151.743
C06099=1101.544,68.449,442.824,176.853,14.590,151.744
C06100=1101.539,68.200,442.841,176.850,14.590,151.745
C06101=1101.533,67.950,442.857,176.848,14.590,151.745
C06102=1101.528,67.701,442.874,176.844,14.589,151.746
C06103=1101.522,67.452,442.891,176.842,14.589,151.746
C06104=1101.517,67.202,442.908,176.840,14.589,151.747
C06105=1101.511,66.953,442.924,176.836,14.588,151.747
C06106=1101.505,66.703,442.941,176.834,14.588,151.748
C06107=1101.499,66.454,442.958,176.832,14.588,151.748
C06108=1101.494,66.205,442.975,176.828,14.588,151.749
C06109=1101.488,65.955,442.991,176.826,14.588,151.749
C06110=1101.482,65.706,443.007,176.824,14.587,151.750
C06111=1101.477,65.456,443.024,176.820,14.587,151.751
C06112=1101.471,65.208,443.041,176.818,14.587,151.751
C06113=1101.465,64.958,443.058,176.816,14.587,151.752
C06114=1101.459,64.709,443.074,176.812,14.586,151.752
C06115=1101.454,64.459,443.091,176.810,14.586,151.753
C06116=1101.447,64.186,443.109,176.807,14.585,151.753
C06117=1101.441,63.914,443.127,176.804,14.586,151.754
C06118=1101.434,63.641,443.145,176.801,14.585,151.754
C06119=1101.428,63.368,443.163,176.799,14.585,151.755
C06120=1101.422,63.120,443.180,176.795,14.585,151.756
C06121=1101.417,62.870,443.196,176.793,14.585,151.756
C06122=1101.411,62.621,443.213,176.791,14.584,151.757
C06123=1101.405,62.371,443.229,176.787,14.584,151.757
C06124=1101.399,62.122,443.245,176.785,14.584,151.758
C06125=1101.394,61.872,443.262,176.783,14.584,151.758
C06126=1101.388,61.623,443.278,176.779,14.583,151.759
C06127=1101.382,61.374,443.295,176.777,14.583,151.759
C06128=1101.376,61.124,443.311,176.775,14.583,151.760
C06129=1101.370,60.875,443.327,176.771,14.583,151.760
C06130=1101.365,60.625,443.344,176.769,14.582,151.761
C06131=1101.359,60.376,443.360,176.767,14.582,151.761
C06132=1101.353,60.127,443.376,176.763,14.582,151.762
C06133=1101.347,59.877,443.393,176.761,14.581,151.762
C06134=1101.342,59.628,443.410,176.759,14.582,151.763
C06135=1101.336,59.378,443.426,176.756,14.581,151.763
C06136=1101.330,59.129,443.442,176.753,14.581,151.764
C06137=1101.324,58.880,443.458,176.751,14.580,151.764
C06138=1101.318,58.630,443.475,176.748,14.580,151.765
C06139=1101.313,58.381,443.491,176.746,14.580,151.765
C06140=1101.307,58.131,443.508,176.743,14.580,151.766
C06141=1101.301,57.882,443.524,176.740,14.579,151.766
C06142=1101.295,57.633,443.540,176.738,14.579,151.767
C06143=1101.289,57.383,443.556,176.735,14.579,151.767
C06144=1101.284,57.135,443.572,176.732,14.578,151.768
C06145=1101.278,56.885,443.589,176.730,14.578,151.768
C06146=1101.273,56.635,443.605,176.727,14.578,151.769
C06147=1101.267,56.386,443.621,176.724,14.577,151.769
C06148=1101.261,56.136,443.637,176.722,14.577,151.770
C06149=1101.255,55.887,443.654,176.720,14.577,151.770
C06150=1101.249,55.637,443.670,176.717,14.577,151.771
C06151=1101.243,55.388,443.686,176.714,14.576,151.772
C06152=1101.238,55.138,443.702,176.712,14.576,151.772
C06153=1101.232,54.889,443.718,176.710,14.576,151.773
C06154=1101.227,54.640,443.734,176.706,14.575,151.773
C06155=1101.221,54.391,443.751,176.704,14.575,151.774
C06156=1101.215,54.141,443.767,176.702,14.575,151.774
C06157=1101.209,53.891,443.782,176.699,14.574,151.775
C06158=1101.203,53.642,443.799,176.696,14.574,151.775
C06159=1101.197,53.393,443.815,176.694,14.574,151.776
C06160=1101.192,53.144,443.831,176.691,14.573,151.776
C06161=1101.187,52.894,443.847,176.689,14.573,151.776
C06162=1101.181,52.644,443.863,176.686,14.573,151.777
C06163=1101.175,52.395,443.879,176.683,14.572,151.777
C06164=1101.169,52.146,443.896,176.681,14.571,151.778
C06165=1101.164,51.896,443.911,176.679,14.572,151.778
C06166=1101.158,51.647,443.927,176.676,14.571,151.779
C06167=1101.152,51.398,443.943,176.673,14.570,151.779
C06168=1101.147,51.148,443.959,176.671,14.570,151.780
C06169=1101.141,50.898,443.975,176.668,14.569,151.780
C06170=1101.135,50.649,443.991,176.666,14.569,151.781
C06171=1101.130,50.400,444.007,176.663,14.569,151.781
C06172=1101.124,50.150,444.023,176.661,14.569,151.782
C06173=1101.118,49.901,444.039,176.658,14.568,151.782
C06174=1101.112,49.651,444.055,176.656,14.568,151.783
C06175=1101.107,49.402,444.071,176.653,14.568,151.783
C06176=1101.101,49.153,444.087,176.650,14.567,151.784
C06177=1101.095,48.903,444.102,176.648,14.567,151.784
C06178=1101.089,48.654,444.119,176.646,14.566,151.784
C06179=1101.084,48.404,444.134,176.643,14.566,151.785
C06180=1101.078,48.131,444.151,176.641,14.565,151.786
C06181=1101.072,47.859,444.169,176.637,14.565,151.786
C06182=1101.066,47.586,444.187,176.635,14.565,151.787
C06183=1101.060,47.313,444.204,176.632,14.564,151.787
C06184=1101.054,47.063,444.219,176.630,14.564,151.788
C06185=1101.048,46.814,444.236,176.628,14.563,151.788
C06186=1101.043,46.565,444.251,176.625,14.562,151.788
C06187=1101.037,46.315,444.267,176.622,14.562,151.789
C06188=1101.031,46.065,444.283,176.620,14.562,151.789
C06189=1101.026,45.816,444.299,176.617,14.561,151.790
C06190=1101.020,45.567,444.314,176.615,14.561,151.790
C06191=1101.015,45.317,444.330,176.613,14.561,151.791
C06192=1101.009,45.067,444.346,176.610,14.560,151.791
C06193=1101.004,44.819,444.362,176.607,14.559,151.792
C06194=1100.998,44.569,444.377,176.605,14.559,151.792
C06195=1100.992,44.319,444.393,176.603,14.559,151.792
C06196=1100.987,44.070,444.409,176.600,14.558,151.793
C06197=1100.981,43.820,444.424,176.598,14.558,151.793
C06198=1100.975,43.571,444.440,176.595,14.558,151.794
C06199=1100.970,43.322,444.455,176.593,14.557,151.794
C06200=1100.964,43.073,444.471,176.590,14.556,151.795
C06201=1100.958,42.823,444.487,176.588,14.556,151.795
C06202=1100.953,42.573,444.502,176.586,14.556,151.796
C06203=1100.946,42.324,444.518,176.583,14.555,151.796
C06204=1100.941,42.074,444.533,176.580,14.555,151.797
C06205=1100.935,41.826,444.549,176.578,14.555,151.797
C06206=1100.930,41.576,444.565,176.576,14.554,151.797
C06207=1100.924,41.326,444.580,176.573,14.553,151.798
C06208=1100.918,41.077,444.595,176.571,14.553,151.798
C06209=1100.912,40.827,444.611,176.569,14.553,151.799
C06210=1100.907,40.578,444.627,176.566,14.552,151.799
C06211=1100.901,40.329,444.642,176.563,14.551,151.800
C06212=1100.895,40.079,444.657,176.561,14.551,151.800
C06213=1100.889,39.829,444.673,176.559,14.551,151.801
C06214=1100.884,39.580,444.688,176.556,14.550,151.801
C06215=1100.878,39.331,444.704,176.554,14.550,151.801
C06216=1100.872,39.081,444.719,176.551,14.550,151.802
C06217=1100.867,38.832,444.734,176.548,14.549,151.802
C06218=1100.861,38.582,444.750,176.546,14.548,151.803
C06219=1100.856,38.333,444.766,176.544,14.548,151.803
C06220=1100.849,38.083,444.781,176.542,14.548,151.804
C06221=1100.844,37.833,444.796,176.539,14.547,151.804
C06222=1100.839,37.584,444.812,176.537,14.546,151.804
C06223=1100.832,37.335,444.827,176.535,14.546,151.805
C06224=1100.827,37.086,444.842,176.532,14.546,151.805
C06225=1100.821,36.836,444.857,176.529,14.545,151.806
C06226=1100.815,36.586,444.873,176.527,14.545,151.806
C06227=1100.810,36.337,444.888,176.525,14.544,151.807
C06228=1100.803,36.088,444.904,176.522,14.543,151.807
C06229=1100.798,35.838,444.919,176.520,14.543,151.807
C06230=1100.792,35.589,444.934,176.518,14.543,151.808
C06231=1100.786,35.339,444.949,176.515,14.542,151.808
C06232=1100.781,35.090,444.965,176.513,14.541,151.809
C06233=1100.775,34.840,444.980,176.510,14.541,151.809
C06234=1100.769,34.590,444.995,176.508,14.541,151.810
C06235=1100.763,34.342,445.010,176.506,14.540,151.810
C06236=1100.757,34.092,445.026,176.503,14.540,151.810
C06237=1100.751,33.843,445.040,176.501,14.539,151.811
C06238=1100.746,33.593,445.056,176.499,14.539,151.811
C06239=1100.740,33.343,445.072,176.496,14.539,151.812
C06240=1100.734,33.094,445.086,176.493,14.538,151.812
C06241=1100.729,32.844,445.102,176.491,14.537,151.813
C06242=1100.723,32.595,445.116,176.489,14.537,151.813
C06243=1100.717,32.345,445.132,176.487,14.537,151.813
C06244=1100.711,32.073,445.148,176.484,14.536,151.814
C06245=1100.704,31.800,445.164,176.482,14.535,151.814
C06246=1100.698,31.527,445.182,176.478,14.535,151.815
C06247=1100.692,31.254,445.198,176.476,14.535,151.815
C06248=1100.686,31.005,445.213,176.474,14.534,151.816
C06249=1100.680,30.755,445.228,176.471,14.533,151.816
C06250=1100.676,30.506,445.243,176.469,14.533,151.816
C06251=1100.669,30.256,445.258,176.467,14.532,151.817
C06252=1100.664,30.007,445.273,176.465,14.532,151.817
C06253=1100.658,29.757,445.288,176.462,14.531,151.818
C06254=1100.652,29.508,445.302,176.460,14.531,151.818
C06255=1100.646,29.258,445.318,176.458,14.530,151.819
C06256=1100.641,29.009,445.333,176.455,14.530,151.819
C06257=1100.635,28.759,445.348,176.452,14.529,151.819
C06258=1100.629,28.510,445.363,176.451,14.528,151.820
C06259=1100.624,28.260,445.378,176.448,14.528,151.820
C06260=1100.618,28.011,445.393,176.446,14.528,151.821
C06261=1100.611,27.762,445.408,176.443,14.527,151.821
C06262=1100.606,27.512,445.423,176.441,14.526,151.821
C06263=1100.600,27.263,445.438,176.439,14.526,151.822
C06264=1100.595,27.013,445.452,176.437,14.526,151.822
C06265=1100.589,26.763,445.467,176.434,14.526,151.823
C06266=1100.583,26.514,445.482,176.432,14.524,151.823
C06267=1100.577,26.264,445.497,176.430,14.524,151.823
C06268=1100.572,26.015,445.512,176.427,14.524,151.824
C06269=1100.565,25.766,445.527,176.425,14.523,151.824
C06270=1100.560,25.516,445.542,176.422,14.522,151.825
C06271=1100.555,25.267,445.556,176.420,14.522,151.825
C06272=1100.548,25.017,445.571,176.418,14.521,151.825
C06273=1100.543,24.768,445.586,176.416,14.521,151.826
C06274=1100.537,24.518,445.601,176.413,14.520,151.826
C06275=1100.531,24.269,445.616,176.411,14.520,151.827
C06276=1100.526,24.019,445.630,176.409,14.519,151.827
C06277=1100.520,23.770,445.645,176.406,14.519,151.827
C06278=1100.514,23.520,445.660,176.405,14.518,151.828
C06279=1100.508,23.271,445.675,176.402,14.517,151.828
C06280=1100.503,23.021,445.689,176.399,14.517,151.829
C06281=1100.497,22.772,445.704,176.397,14.517,151.829
C06282=1100.491,22.523,445.719,176.395,14.516,151.829
C06283=1100.485,22.273,445.734,176.393,14.516,151.830
C06284=1100.480,22.023,445.748,176.390,14.515,151.830
C06285=1100.473,21.773,445.763,176.388,14.514,151.831
C06286=1100.468,21.524,445.777,176.386,14.514,151.831
C06287=1100.463,21.275,445.792,176.384,14.513,151.831
C06288=1100.457,21.025,445.807,176.381,14.512,151.832
C06289=1100.451,20.776,445.821,176.379,14.512,151.832
C06290=1100.445,20.526,445.835,176.377,14.511,151.832
C06291=1100.440,20.276,445.851,176.375,14.511,151.833
C06292=1100.434,20.027,445.865,176.373,14.511,151.833
C06293=1100.428,19.777,445.880,176.370,14.510,151.834
C06294=1100.422,19.528,445.894,176.368,14.509,151.834
C06295=1100.416,19.279,445.909,176.366,14.509,151.834
C06296=1100.410,19.029,445.923,176.363,14.508,151.835
C06297=1100.405,18.780,445.938,176.361,14.508,151.835
C06298=1100.399,18.529,445.952,176.359,14.507,151.835
C06299=1100.393,18.280,445.967,176.356,14.506,151.836
C06300=1100.387,18.032,445.982,176.354,14.506,151.836
C06301=1100.381,17.781,445.996,176.352,14.506,151.837
C06302=1100.376,17.532,446.010,176.350,14.505,151.837
C06303=1100.370,17.283,446.024,176.347,14.504,151.837
C06304=1100.364,17.033,446.040,176.345,14.504,151.838
C06305=1100.359,16.783,446.054,176.343,14.503,151.838
C06306=1100.353,16.534,446.068,176.341,14.503,151.838
C06307=1100.347,16.284,446.083,176.339,14.502,151.839
C06308=1100.341,16.013,446.098,176.336,14.501,151.839
C06309=1100.335,15.742,446.114,176.334,14.500,151.840
C06310=1100.328,15.470,446.130,176.331,14.500,151.840
C06311=1100.322,15.199,446.145,176.329,14.499,151.841
C06312=1100.317,14.949,446.160,176.326,14.499,151.841
C06313=1100.311,14.700,446.175,176.325,14.498,151.841
C06314=1100.305,14.450,446.188,176.322,14.498,151.842
C06315=1100.299,14.201,446.203,176.319,14.497,151.842
C06316=1100.293,13.951,446.217,176.318,14.496,151.842
C06317=1100.288,13.702,446.232,176.315,14.496,151.843
C06318=1100.282,13.452,446.246,176.313,14.496,151.843
C06319=1100.276,13.202,446.260,176.311,14.495,151.843
C06320=1100.270,12.954,446.274,176.308,14.494,151.844
C06321=1100.263,12.703,446.288,176.306,14.494,151.844
C06322=1100.258,12.454,446.303,176.304,14.493,151.845
C06323=1100.252,12.205,446.317,176.302,14.492,151.845
C06324=1100.246,11.955,446.331,176.300,14.492,151.845
C06325=1100.240,11.706,446.345,176.298,14.491,151.846
C06326=1100.235,11.456,446.359,176.295,14.490,151.846
C06327=1100.229,11.206,446.374,176.293,14.490,151.847
C06328=1100.223,10.957,446.388,176.291,14.489,151.847
C06329=1100.218,10.707,446.402,176.289,14.489,151.847
C06330=1100.212,10.458,446.416,176.287,14.489,151.848
C06331=1100.206,10.208,446.431,176.285,14.488,151.848
C06332=1100.199,9.959,446.444,176.282,14.487,151.848
C06333=1100.194,9.710,446.459,176.280,14.486,151.849
C06334=1100.188,9.459,446.473,176.278,14.486,151.849
C06335=1100.182,9.210,446.487,176.276,14.486,151.849
C06336=1100.176,8.961,446.501,176.274,14.485,151.850
C06337=1100.171,8.711,446.515,176.271,14.485,151.850
C06338=1100.165,8.461,446.529,176.269,14.483,151.850
C06339=1100.159,8.212,446.544,176.267,14.483,151.851
C06340=1100.154,7.963,446.558,176.264,14.483,151.851
C06341=1100.147,7.713,446.571,176.263,14.482,151.852
C06342=1100.141,7.463,446.585,176.260,14.481,151.852
C06343=1100.135,7.214,446.600,176.259,14.481,151.852
C06344=1100.130,6.964,446.614,176.256,14.480,151.853
C06345=1100.125,6.715,446.628,176.254,14.479,151.853
C06346=1100.118,6.465,446.642,176.252,14.479,151.853
C06347=1100.112,6.216,446.656,176.249,14.478,151.854
C06348=1100.106,5.966,446.670,176.247,14.478,151.854
C06349=1100.101,5.717,446.684,176.245,14.477,151.854
C06350=1100.096,5.467,446.697,176.243,14.477,151.855
C06351=1100.089,5.217,446.712,176.240,14.476,151.855
C06352=1100.084,4.967,446.725,176.239,14.475,151.855
C06353=1100.077,4.719,446.739,176.236,14.475,151.856
C06354=1100.072,4.469,446.753,176.234,14.474,151.856
C06355=1100.066,4.220,446.767,176.232,14.473,151.856
C06356=1100.060,3.969,446.781,176.230,14.473,151.857
C06357=1100.055,3.720,446.795,176.228,14.472,151.857
C06358=1100.049,3.470,446.809,176.226,14.471,151.857
C06359=1100.043,3.221,446.822,176.223,14.471,151.858
C06360=1100.037,2.972,446.837,176.222,14.470,151.858
C06361=1100.032,2.722,446.851,176.219,14.470,151.859
C06362=1100.026,2.473,446.865,176.217,14.469,151.859
C06363=1100.020,2.223,446.878,176.215,14.469,151.859
C06364=1100.014,1.973,446.892,176.213,14.467,151.860
C06365=1100.009,1.724,446.906,176.210,14.467,151.860
C06366=1100.003,1.474,446.920,176.209,14.466,151.860
C06367=1099.997,1.225,446.933,176.206,14.466,151.861
C06368=1099.992,0.975,446.947,176.204,14.465,151.861
C06369=1099.986,0.726,446.961,176.202,14.465,151.861
C06370=1099.981,0.476,446.975,176.200,14.464,151.862
C06371=1099.974,0.226,446.988,176.199,14.463,151.862
C06372=1099.968,-0.043,447.004,176.196,14.462,151.862
C06373=1099.962,-0.312,447.018,176.193,14.462,151.863
C06374=1099.956,-0.581,447.033,176.192,14.461,151.863
C06375=1099.950,-0.851,447.048,176.189,14.460,151.863
C06376=1099.944,-1.101,447.062,176.187,14.459,151.864
C06377=1099.938,-1.350,447.075,176.185,14.459,151.864
C06378=1099.933,-1.600,447.089,176.183,14.458,151.864
C06379=1099.927,-1.849,447.103,176.181,14.458,151.865
C06380=1099.921,-2.098,447.116,176.179,14.457,151.865
C06381=1099.915,-2.349,447.130,176.177,14.457,151.865
C06382=1099.910,-2.598,447.144,176.174,14.456,151.866
C06383=1099.904,-2.848,447.158,176.172,14.455,151.866
C06384=1099.898,-3.097,447.171,176.170,14.454,151.866
C06385=1099.892,-3.347,447.185,176.168,14.454,151.867
C06386=1099.886,-3.597,447.198,176.166,14.453,151.867
C06387=1099.881,-3.846,447.212,176.164,14.453,151.867
C06388=1099.875,-4.096,447.226,176.162,14.452,151.868
C06389=1099.869,-4.345,447.239,176.160,14.452,151.868
C06390=1099.864,-4.595,447.253,176.157,14.450,151.868
C06391=1099.858,-4.844,447.266,176.155,14.450,151.869
C06392=1099.852,-5.094,447.280,176.153,14.449,151.869
C06393=1099.845,-5.343,447.294,176.151,14.448,151.869
C06394=1099.840,-5.593,447.307,176.149,14.448,151.870
C06395=1099.834,-5.843,447.320,176.147,14.447,151.870
C06396=1099.828,-6.092,447.334,176.145,14.447,151.870
C06397=1099.822,-6.342,447.347,176.143,14.446,151.871
C06398=1099.817,-6.591,447.361,176.141,14.446,151.871
C06399=1099.811,-6.841,447.374,176.139,14.445,151.871
C06400=1099.805,-7.090,447.388,176.136,14.444,151.872
C06401=1099.799,-7.340,447.401,176.134,14.444,151.872
C06402=1099.794,-7.590,447.414,176.132,14.443,151.872
C06403=1099.787,-7.839,447.428,176.130,14.442,151.873
C06404=1099.781,-8.088,447.441,176.128,14.442,151.873
C06405=1099.776,-8.338,447.455,176.126,14.441,151.873
C06406=1099.770,-8.588,447.467,176.124,14.441,151.874
C06407=1099.764,-8.837,447.481,176.122,14.440,151.874
C06408=1099.758,-9.086,447.495,176.120,14.440,151.874
C06409=1099.753,-9.336,447.508,176.118,14.439,151.875
C06410=1099.746,-9.587,447.521,176.115,14.437,151.875
C06411=1099.741,-9.836,447.535,176.113,14.437,151.875
C06412=1099.734,-10.085,447.548,176.111,14.436,151.876
C06413=1099.729,-10.335,447.561,176.109,14.436,151.876
C06414=1099.723,-10.585,447.575,176.107,14.435,151.876
C06415=1099.717,-10.834,447.588,176.105,14.435,151.877
C06416=1099.711,-11.084,447.602,176.103,14.434,151.877
C06417=1099.705,-11.334,447.615,176.101,14.433,151.877
C06418=1099.701,-11.582,447.628,176.100,14.433,151.877
C06419=1099.694,-11.832,447.641,176.097,14.432,151.878
C06420=1099.689,-12.082,447.654,176.095,14.432,151.878
C06421=1099.683,-12.331,447.668,176.094,14.431,151.878
C06422=1099.677,-12.581,447.680,176.091,14.430,151.879
C06423=1099.672,-12.831,447.694,176.089,14.429,151.879
C06424=1099.665,-13.080,447.707,176.087,14.428,151.879
C06425=1099.660,-13.330,447.720,176.085,14.428,151.880
C06426=1099.654,-13.579,447.734,176.083,14.427,151.880
C06427=1099.648,-13.829,447.747,176.081,14.427,151.880
C06428=1099.643,-14.079,447.760,176.079,14.426,151.881
C06429=1099.636,-14.328,447.774,176.077,14.426,151.881
C06430=1099.631,-14.578,447.786,176.075,14.425,151.881
C06431=1099.625,-14.828,447.800,176.073,14.424,151.882
C06432=1099.619,-15.077,447.813,176.071,14.424,151.882
C06433=1099.613,-15.327,447.826,176.069,14.423,151.882
C06434=1099.607,-15.576,447.840,176.067,14.423,151.883
C06435=1099.602,-15.826,447.852,176.064,14.421,151.883
C06436=1099.595,-16.093,447.866,176.062,14.420,151.883
C06437=1099.589,-16.361,447.880,176.060,14.420,151.884
C06438=1099.582,-16.629,447.894,176.058,14.419,151.884
C06439=1099.576,-16.897,447.909,176.056,14.419,151.884
C06440=1099.570,-17.146,447.922,176.054,14.418,151.885
C06441=1099.564,-17.396,447.934,176.052,14.418,151.885
C06442=1099.559,-17.645,447.947,176.049,14.417,151.885
C06443=1099.553,-17.895,447.960,176.048,14.416,151.886
C06444=1099.547,-18.144,447.974,176.045,14.416,151.886
C06445=1099.541,-18.394,447.986,176.043,14.415,151.886
C06446=1099.535,-18.644,447.999,176.042,14.414,151.886
C06447=1099.529,-18.893,448.012,176.039,14.414,151.887
C06448=1099.523,-19.143,448.025,176.038,14.413,151.887
C06449=1099.518,-19.393,448.038,176.036,14.412,151.887
C06450=1099.512,-19.643,448.051,176.034,14.412,151.888
C06451=1099.506,-19.892,448.064,176.032,14.411,151.888
C06452=1099.500,-20.142,448.077,176.030,14.410,151.888
C06453=1099.494,-20.391,448.090,176.028,14.410,151.889
C06454=1099.489,-20.641,448.103,176.026,14.409,151.889
C06455=1099.483,-20.890,448.115,176.024,14.409,151.889
C06456=1099.477,-21.140,448.129,176.022,14.408,151.890
C06457=1099.471,-21.390,448.141,176.020,14.408,151.890
C06458=1099.465,-21.639,448.155,176.018,14.407,151.890
C06459=1099.459,-21.889,448.167,176.016,14.406,151.891
C06460=1099.453,-22.139,448.180,176.014,14.406,151.891
C06461=1099.447,-22.388,448.193,176.012,14.405,151.891
C06462=1099.442,-22.637,448.206,176.010,14.404,151.891
C06463=1099.436,-22.887,448.218,176.008,14.403,151.892
C06464=1099.430,-23.137,448.232,176.006,14.403,151.892
C06465=1099.424,-23.386,448.244,176.003,14.402,151.892
C06466=1099.418,-23.636,448.257,176.001,14.401,151.893
C06467=1099.412,-23.886,448.270,176.000,14.400,151.893
C06468=1099.407,-24.135,448.283,175.997,14.400,151.893
C06469=1099.402,-24.385,448.295,175.995,14.399,151.894
C06470=1099.395,-24.634,448.308,175.994,14.398,151.894
C06471=1099.389,-24.884,448.321,175.992,14.398,151.894
C06472=1099.384,-25.134,448.334,175.990,14.397,151.895
C06473=1099.378,-25.383,448.346,175.988,14.397,151.895
C06474=1099.372,-25.632,448.359,175.986,14.396,151.895
C06475=1099.366,-25.882,448.372,175.984,14.395,151.895
C06476=1099.360,-26.132,448.384,175.982,14.395,151.896
C06477=1099.354,-26.382,448.397,175.980,14.394,151.896
C06478=1099.349,-26.631,448.410,175.978,14.393,151.896
C06479=1099.343,-26.881,448.423,175.976,14.393,151.897
C06480=1099.338,-27.131,448.435,175.974,14.392,151.897
C06481=1099.332,-27.381,448.448,175.972,14.391,151.897
C06482=1099.325,-27.630,448.461,175.970,14.391,151.898
C06483=1099.319,-27.879,448.473,175.968,14.390,151.898
C06484=1099.313,-28.129,448.485,175.966,14.390,151.898
C06485=1099.308,-28.378,448.498,175.964,14.389,151.898
C06486=1099.302,-28.628,448.510,175.962,14.388,151.899
C06487=1099.296,-28.878,448.523,175.960,14.388,151.899
C06488=1099.290,-29.128,448.536,175.958,14.387,151.899
C06489=1099.284,-29.377,448.548,175.956,14.386,151.900
C06490=1099.278,-29.627,448.561,175.954,14.386,151.900
C06491=1099.272,-29.876,448.574,175.952,14.385,151.900
C06492=1099.267,-30.126,448.586,175.950,14.385,151.901
C06493=1099.261,-30.376,448.599,175.949,14.384,151.901
C06494=1099.255,-30.625,448.612,175.946,14.383,151.901
C06495=1099.248,-30.874,448.623,175.945,14.383,151.902
C06496=1099.242,-31.124,448.636,175.943,14.382,151.902
C06497=1099.237,-31.374,448.649,175.941,14.381,151.902
C06498=1099.231,-31.623,448.661,175.939,14.381,151.903
C06499=1099.225,-31.873,448.673,175.937,14.380,151.903
C06500=1099.219,-32.141,448.687,175.935,14.379,151.903
C06501=1099.212,-32.408,448.700,175.933,14.379,151.903
C06502=1099.207,-32.674,448.714,175.931,14.378,151.904
C06503=1099.200,-32.941,448.727,175.929,14.378,151.904
C06504=1099.194,-33.191,448.739,175.927,14.377,151.904
C06505=1099.188,-33.440,448.751,175.925,14.376,151.905
C06506=1099.183,-33.690,448.764,175.923,14.376,151.905
C06507=1099.177,-33.940,448.777,175.921,14.375,151.905
C06508=1099.171,-34.189,448.788,175.919,14.375,151.906
C06509=1099.165,-34.439,448.801,175.917,14.374,151.906
C06510=1099.159,-34.689,448.813,175.915,14.373,151.906
C06511=1099.153,-34.938,448.826,175.913,14.372,151.906
C06512=1099.148,-35.188,448.838,175.911,14.372,151.907
C06513=1099.142,-35.438,448.851,175.909,14.371,151.907
C06514=1099.136,-35.687,448.863,175.907,14.371,151.907
C06515=1099.130,-35.936,448.875,175.905,14.370,151.908
C06516=1099.124,-36.186,448.887,175.904,14.369,151.908
C06517=1099.118,-36.436,448.900,175.901,14.369,151.908
C06518=1099.113,-36.685,448.912,175.900,14.368,151.909
C06519=1099.107,-36.935,448.925,175.898,14.367,151.909
C06520=1099.100,-37.185,448.937,175.896,14.367,151.909
C06521=1099.095,-37.434,448.949,175.894,14.366,151.909
C06522=1099.089,-37.684,448.961,175.892,14.365,151.910
C06523=1099.083,-37.934,448.974,175.890,14.365,151.910
C06524=1099.078,-38.183,448.986,175.888,14.364,151.910
C06525=1099.071,-38.433,448.997,175.886,14.363,151.911
C06526=1099.065,-38.683,449.010,175.884,14.362,151.911
C06527=1099.060,-38.932,449.022,175.882,14.362,151.911
C06528=1099.054,-39.182,449.035,175.880,14.361,151.912
C06529=1099.048,-39.432,449.047,175.878,14.361,151.912
C06530=1099.042,-39.681,449.059,175.876,14.360,151.912
C06531=1099.036,-39.931,449.071,175.875,14.360,151.912
C06532=1099.030,-40.180,449.083,175.873,14.359,151.913
C06533=1099.024,-40.430,449.096,175.871,14.359,151.913
C06534=1099.019,-40.680,449.107,175.869,14.358,151.913
C06535=1099.012,-40.929,449.119,175.867,14.358,151.914
C06536=1099.006,-41.179,449.132,175.865,14.357,151.914
C06537=1099.000,-41.428,449.143,175.863,14.356,151.914
C06538=1098.994,-41.678,449.156,175.862,14.355,151.914
C06539=1098.988,-41.928,449.168,175.859,14.355,151.915
C06540=1098.983,-42.177,449.179,175.857,14.354,151.915
C06541=1098.977,-42.427,449.192,175.856,14.354,151.915
C06542=1098.971,-42.677,449.204,175.854,14.353,151.916
C06543=1098.965,-42.926,449.216,175.851,14.353,151.916
C06544=1098.959,-43.176,449.229,175.850,14.352,151.916
C06545=1098.953,-43.425,449.239,175.848,14.351,151.917
C06546=1098.947,-43.675,449.252,175.846,14.350,151.917
C06547=1098.941,-43.925,449.265,175.844,14.351,151.917
C06548=1098.935,-44.174,449.276,175.843,14.350,151.918
C06549=1098.930,-44.425,449.288,175.841,14.349,151.918
C06550=1098.923,-44.674,449.300,175.839,14.348,151.918
C06551=1098.918,-44.923,449.312,175.837,14.348,151.918
C06552=1098.911,-45.173,449.324,175.835,14.347,151.919
C06553=1098.906,-45.423,449.336,175.833,14.347,151.919
C06554=1098.900,-45.673,449.348,175.831,14.346,151.919
C06555=1098.893,-45.922,449.360,175.829,14.345,151.920
C06556=1098.888,-46.172,449.372,175.827,14.344,151.920
C06557=1098.882,-46.422,449.384,175.825,14.344,151.920
C06558=1098.876,-46.671,449.396,175.823,14.343,151.921
C06559=1098.870,-46.920,449.408,175.821,14.342,151.921
C06560=1098.865,-47.170,449.419,175.820,14.342,151.921
C06561=1098.859,-47.420,449.432,175.818,14.342,151.921
C06562=1098.852,-47.670,449.444,175.816,14.341,151.922
C06563=1098.847,-47.919,449.455,175.814,14.341,151.922
C06564=1098.841,-48.187,449.468,175.812,14.340,151.922
C06565=1098.834,-48.453,449.480,175.810,14.339,151.923
C06566=1098.828,-48.721,449.493,175.808,14.339,151.923
C06567=1098.822,-48.989,449.506,175.806,14.338,151.923
C06568=1098.816,-49.238,449.517,175.805,14.337,151.923
C06569=1098.810,-49.488,449.530,175.803,14.336,151.924
C06570=1098.804,-49.737,449.541,175.800,14.336,151.924
C06571=1098.798,-49.987,449.553,175.799,14.335,151.924
C06572=1098.793,-50.236,449.564,175.797,14.335,151.925
C06573=1098.787,-50.486,449.577,175.795,14.334,151.925
C06574=1098.781,-50.736,449.588,175.793,14.333,151.925
C06575=1098.775,-50.986,449.600,175.791,14.333,151.926
C06576=1098.768,-51.235,449.612,175.790,14.333,151.926
C06577=1098.763,-51.485,449.623,175.788,14.332,151.926
C06578=1098.757,-51.735,449.636,175.786,14.332,151.927
C06579=1098.750,-51.985,449.647,175.784,14.331,151.927
C06580=1098.744,-52.234,449.658,175.782,14.330,151.927
C06581=1098.739,-52.484,449.670,175.780,14.329,151.927
C06582=1098.733,-52.733,449.682,175.778,14.329,151.928
C06583=1098.726,-52.983,449.694,175.776,14.328,151.928
C06584=1098.720,-53.232,449.705,175.775,14.328,151.928
C06585=1098.714,-53.482,449.717,175.773,14.328,151.929
C06586=1098.708,-53.732,449.729,175.771,14.327,151.929
C06587=1098.702,-53.981,449.740,175.769,14.326,151.929
C06588=1098.696,-54.232,449.752,175.767,14.326,151.929
C06589=1098.690,-54.480,449.764,175.765,14.325,151.930
C06590=1098.684,-54.731,449.775,175.763,14.325,151.930
C06591=1098.678,-54.979,449.786,175.762,14.325,151.930
C06592=1098.672,-55.230,449.798,175.760,14.324,151.931
C06593=1098.666,-55.479,449.810,175.758,14.324,151.931
C06594=1098.660,-55.729,449.821,175.756,14.323,151.931
C06595=1098.654,-55.979,449.832,175.754,14.322,151.932
C06596=1098.648,-56.228,449.844,175.752,14.321,151.932
C06597=1098.642,-56.479,449.856,175.750,14.321,151.932
C06598=1098.636,-56.727,449.867,175.749,14.321,151.933
C06599=1098.630,-56.978,449.879,175.747,14.320,151.933
C06600=1098.624,-57.227,449.891,175.745,14.320,151.933
C06601=1098.618,-57.477,449.902,175.743,14.319,151.933
C06602=1098.612,-57.727,449.913,175.741,14.318,151.934
C06603=1098.606,-57.976,449.925,175.739,14.318,151.934
C06604=1098.601,-58.226,449.936,175.737,14.317,151.934
C06605=1098.594,-58.475,449.948,175.736,14.317,151.935
C06606=1098.588,-58.725,449.959,175.734,14.316,151.935
C06607=1098.582,-58.974,449.970,175.732,14.316,151.935
C06608=1098.576,-59.224,449.982,175.730,14.315,151.936
C06609=1098.571,-59.474,449.993,175.728,14.315,151.936
C06610=1098.564,-59.724,450.005,175.726,14.314,151.936
C06611=1098.558,-59.973,450.016,175.725,14.314,151.936
C06612=1098.552,-60.223,450.028,175.723,14.313,151.937
C06613=1098.546,-60.473,450.038,175.721,14.313,151.937
C06614=1098.540,-60.722,450.051,175.719,14.312,151.937
C06615=1098.535,-60.972,450.062,175.717,14.311,151.938
C06616=1098.528,-61.222,450.073,175.715,14.311,151.938
C06617=1098.522,-61.471,450.085,175.713,14.310,151.938
C06618=1098.516,-61.721,450.096,175.712,14.310,151.939
C06619=1098.510,-61.971,450.107,175.710,14.309,151.939
C06620=1098.505,-62.220,450.119,175.708,14.309,151.939
C06621=1098.499,-62.470,450.130,175.706,14.308,151.939
C06622=1098.493,-62.720,450.141,175.704,14.307,151.940
C06623=1098.486,-62.970,450.152,175.703,14.307,151.940
C06624=1098.480,-63.219,450.164,175.701,14.307,151.940
C06625=1098.475,-63.468,450.175,175.699,14.306,151.941
C06626=1098.469,-63.719,450.187,175.697,14.306,151.941
C06627=1098.463,-63.968,450.198,175.695,14.305,151.941
C06628=1098.456,-64.237,450.210,175.693,14.305,151.942
C06629=1098.450,-64.505,450.222,175.691,14.304,151.942
C06630=1098.444,-64.774,450.235,175.689,14.303,151.942
C06631=1098.437,-65.042,450.246,175.687,14.303,151.943
C06632=1098.432,-65.292,450.257,175.686,14.303,151.943
C06633=1098.425,-65.542,450.269,175.684,14.302,151.943
C06634=1098.419,-65.791,450.279,175.682,14.301,151.943
C06635=1098.413,-66.042,450.291,175.680,14.300,151.944
C06636=1098.408,-66.291,450.303,175.678,14.300,151.944
C06637=1098.402,-66.540,450.314,175.677,14.300,151.944
C06638=1098.396,-66.790,450.325,175.675,14.299,151.945
C06639=1098.390,-67.040,450.336,175.673,14.298,151.945
C06640=1098.384,-67.289,450.347,175.671,14.298,151.945
C06641=1098.378,-67.540,450.358,175.669,14.297,151.945
C06642=1098.372,-67.789,450.369,175.668,14.297,151.946
C06643=1098.366,-68.038,450.380,175.666,14.297,151.946
C06644=1098.360,-68.288,450.392,175.664,14.296,151.946
C06645=1098.354,-68.538,450.403,175.662,14.296,151.947
C06646=1098.349,-68.787,450.414,175.660,14.295,151.947
C06647=1098.343,-69.038,450.425,175.659,14.295,151.947
C06648=1098.337,-69.287,450.436,175.657,14.294,151.947
C06649=1098.331,-69.537,450.447,175.655,14.294,151.948
C06650=1098.325,-69.787,450.458,175.653,14.293,151.948
C06651=1098.319,-70.036,450.469,175.651,14.292,151.948
C06652=1098.313,-70.286,450.480,175.650,14.292,151.949
C06653=1098.307,-70.535,450.492,175.648,14.292,151.949
C06654=1098.301,-70.785,450.503,175.646,14.291,151.949
C06655=1098.295,-71.034,450.514,175.644,14.290,151.950
C06656=1098.290,-71.284,450.525,175.643,14.290,151.950
C06657=1098.283,-71.534,450.536,175.641,14.290,151.950
C06658=1098.278,-71.784,450.547,175.639,14.289,151.950
C06659=1098.272,-72.033,450.558,175.637,14.288,151.951
C06660=1098.266,-72.282,450.568,175.635,14.288,151.951
C06661=1098.260,-72.533,450.580,175.634,14.287,151.951
C06662=1098.255,-72.782,450.591,175.632,14.287,151.952
C06663=1098.249,-73.032,450.602,175.630,14.286,151.952
C06664=1098.243,-73.282,450.613,175.628,14.286,151.952
C06665=1098.237,-73.532,450.624,175.627,14.286,151.952
C06666=1098.231,-73.781,450.635,175.625,14.285,151.953
C06667=1098.225,-74.031,450.646,175.623,14.285,151.953
C06668=1098.219,-74.281,450.657,175.621,14.284,151.953
C06669=1098.213,-74.530,450.668,175.620,14.284,151.954
C06670=1098.207,-74.779,450.678,175.618,14.283,151.954
C06671=1098.201,-75.029,450.689,175.616,14.283,151.954
C06672=1098.195,-75.280,450.700,175.614,14.282,151.955
C06673=1098.189,-75.529,450.711,175.612,14.282,151.955
C06674=1098.184,-75.779,450.722,175.611,14.281,151.955
C06675=1098.177,-76.029,450.733,175.609,14.281,151.956
C06676=1098.171,-76.278,450.744,175.607,14.280,151.956
C06677=1098.165,-76.528,450.754,175.606,14.280,151.956
C06678=1098.159,-76.777,450.765,175.604,14.280,151.956
C06679=1098.153,-77.027,450.776,175.602,14.279,151.957
C06680=1098.147,-77.277,450.787,175.600,14.279,151.957
C06681=1098.141,-77.526,450.798,175.599,14.278,151.957
C06682=1098.135,-77.776,450.809,175.597,14.278,151.958
C06683=1098.129,-78.026,450.819,175.595,14.277,151.958
C06684=1098.123,-78.276,450.829,175.593,14.277,151.958
C06685=1098.117,-78.525,450.840,175.591,14.277,151.959
C06686=1098.111,-78.775,450.852,175.590,14.276,151.959
C06687=1098.105,-79.025,450.862,175.587,14.276,151.959
C06688=1098.100,-79.274,450.873,175.586,14.275,151.960
C06689=1098.093,-79.524,450.884,175.584,14.275,151.960
C06690=1098.087,-79.774,450.895,175.582,14.274,151.960
C06691=1098.081,-80.024,450.905,175.580,14.274,151.960
C06692=1098.075,-80.295,450.917,175.578,14.273,151.961
C06693=1098.068,-80.565,450.928,175.577,14.273,151.961
C06694=1098.062,-80.836,450.941,175.575,14.272,151.961
C06695=1098.055,-81.107,450.952,175.573,14.272,151.962
C06696=1098.049,-81.356,450.963,175.571,14.271,151.962
C06697=1098.042,-81.606,450.973,175.569,14.271,151.962
C06698=1098.037,-81.856,450.983,175.568,14.271,151.963
C06699=1098.031,-82.106,450.994,175.566,14.270,151.963
C06700=1098.024,-82.355,451.005,175.564,14.270,151.963
C06701=1098.018,-82.605,451.015,175.563,14.270,151.964
C06702=1098.013,-82.854,451.026,175.561,14.269,151.964
C06703=1098.006,-83.105,451.036,175.558,14.269,151.964
C06704=1098.000,-83.354,451.047,175.557,14.268,151.965
C06705=1097.994,-83.604,451.058,175.556,14.268,151.965
C06706=1097.988,-83.853,451.068,175.553,14.268,151.965
C06707=1097.982,-84.104,451.079,175.551,14.267,151.966
C06708=1097.976,-84.353,451.089,175.550,14.267,151.966
C06709=1097.970,-84.602,451.100,175.548,14.267,151.966
C06710=1097.964,-84.852,451.111,175.546,14.266,151.966
C06711=1097.957,-85.102,451.121,175.545,14.266,151.967
C06712=1097.952,-85.352,451.132,175.543,14.266,151.967
C06713=1097.945,-85.601,451.142,175.541,14.265,151.967
C06714=1097.940,-85.851,451.152,175.540,14.265,151.968
C06715=1097.934,-86.101,451.163,175.538,14.264,151.968
C06716=1097.927,-86.350,451.174,175.536,14.264,151.968
C06717=1097.921,-86.601,451.184,175.534,14.264,151.969
C06718=1097.916,-86.850,451.195,175.533,14.263,151.969
C06719=1097.909,-87.099,451.205,175.530,14.263,151.969
C06720=1097.904,-87.349,451.215,175.528,14.262,151.970
C06721=1097.897,-87.599,451.226,175.527,14.262,151.970
C06722=1097.891,-87.849,451.237,175.525,14.262,151.970
C06723=1097.885,-88.098,451.246,175.523,14.261,151.971
C06724=1097.879,-88.348,451.257,175.522,14.261,151.971
C06725=1097.873,-88.597,451.268,175.520,14.261,151.971
C06726=1097.867,-88.847,451.278,175.518,14.260,151.972
C06727=1097.861,-89.097,451.289,175.517,14.260,151.972
C06728=1097.854,-89.347,451.299,175.515,14.260,151.972
C06729=1097.849,-89.597,451.309,175.513,14.259,151.972
C06730=1097.842,-89.846,451.320,175.511,14.259,151.973
C06731=1097.837,-90.096,451.330,175.510,14.258,151.973
C06732=1097.831,-90.345,451.341,175.508,14.258,151.973
C06733=1097.825,-90.595,451.351,175.506,14.258,151.974
C06734=1097.819,-90.845,451.361,175.504,14.257,151.974
C06735=1097.812,-91.095,451.372,175.502,14.257,151.975
C06736=1097.807,-91.345,451.382,175.501,14.257,151.975
C06737=1097.800,-91.594,451.392,175.499,14.256,151.975
C06738=1097.795,-91.844,451.402,175.498,14.257,151.975
C06739=1097.788,-92.093,451.413,175.496,14.256,151.976
C06740=1097.783,-92.343,451.423,175.494,14.256,151.976
C06741=1097.776,-92.593,451.433,175.493,14.255,151.976
C06742=1097.770,-92.843,451.444,175.491,14.255,151.977
C06743=1097.764,-93.093,451.454,175.488,14.254,151.977
C06744=1097.758,-93.342,451.465,175.487,14.254,151.977
C06745=1097.753,-93.592,451.475,175.485,14.254,151.978
C06746=1097.746,-93.841,451.485,175.483,14.253,151.978
C06747=1097.741,-94.091,451.495,175.482,14.253,151.978
C06748=1097.735,-94.341,451.505,175.480,14.253,151.979
C06749=1097.729,-94.591,451.516,175.478,14.252,151.979
C06750=1097.723,-94.840,451.525,175.477,14.252,151.979
C06751=1097.717,-95.090,451.536,175.475,14.252,151.980
C06752=1097.711,-95.340,451.546,175.474,14.252,151.980
C06753=1097.705,-95.590,451.557,175.471,14.251,151.980
C06754=1097.698,-95.840,451.567,175.470,14.251,151.980
C06755=1097.693,-96.089,451.577,175.468,14.250,151.981
C06756=1097.686,-96.362,451.588,175.466,14.250,151.981
C06757=1097.680,-96.635,451.599,175.464,14.249,151.981
C06758=1097.673,-96.908,451.611,175.462,14.249,151.982
C06759=1097.667,-97.182,451.621,175.461,14.249,151.982
C06760=1097.660,-97.431,451.632,175.459,14.249,151.982
C06761=1097.654,-97.681,451.641,175.457,14.248,151.983
C06762=1097.648,-97.930,451.652,175.456,14.248,151.983
C06763=1097.642,-98.180,451.662,175.454,14.248,151.983
C06764=1097.637,-98.430,451.672,175.451,14.247,151.984
C06765=1097.630,-98.679,451.682,175.450,14.247,151.984
C06766=1097.624,-98.930,451.692,175.448,14.247,151.985
C06767=1097.617,-99.179,451.702,175.447,14.247,151.985
C06768=1097.612,-99.429,451.713,175.445,14.246,151.985
C06769=1097.606,-99.679,451.722,175.443,14.246,151.985
C06770=1097.599,-99.928,451.732,175.442,14.246,151.986
C06771=1097.594,-100.178,451.743,175.440,14.246,151.986
C06772=1097.587,-100.428,451.752,175.439,14.245,151.986
C06773=1097.581,-100.677,451.762,175.436,14.245,151.987
C06774=1097.576,-100.927,451.773,175.434,14.244,151.987
C06775=1097.569,-101.177,451.782,175.433,14.245,151.987
C06776=1097.563,-101.426,451.792,175.431,14.244,151.988
C06777=1097.557,-101.676,451.803,175.430,14.244,151.988
C06778=1097.551,-101.926,451.812,175.428,14.244,151.988
C06779=1097.545,-102.175,451.822,175.426,14.244,151.989
C06780=1097.538,-102.426,451.832,175.425,14.243,151.989
C06781=1097.533,-102.676,451.843,175.422,14.243,151.989
C06782=1097.526,-102.925,451.853,175.421,14.243,151.990
C06783=1097.520,-103.175,451.862,175.419,14.243,151.990
C06784=1097.514,-103.424,451.872,175.418,14.243,151.990
C06785=1097.508,-103.675,451.882,175.416,14.242,151.991
C06786=1097.502,-103.924,451.892,175.414,14.242,151.991
C06787=1097.496,-104.174,451.902,175.412,14.242,151.991
C06788=1097.490,-104.423,451.912,175.410,14.241,151.992
C06789=1097.484,-104.673,451.922,175.409,14.242,151.992
C06790=1097.478,-104.923,451.932,175.407,14.241,151.992
C06791=1097.471,-105.172,451.942,175.406,14.241,151.993
C06792=1097.465,-105.422,451.951,175.404,14.240,151.993
C06793=1097.460,-105.672,451.962,175.402,14.240,151.993
C06794=1097.453,-105.922,451.972,175.401,14.240,151.994
C06795=1097.447,-106.171,451.981,175.398,14.240,151.994
C06796=1097.441,-106.421,451.991,175.397,14.240,151.994
C06797=1097.436,-106.671,452.001,175.395,14.239,151.995
C06798=1097.429,-106.920,452.011,175.394,14.239,151.995
C06799=1097.423,-107.170,452.021,175.392,14.239,151.995
C06800=1097.417,-107.420,452.030,175.391,14.239,151.996
C06801=1097.411,-107.670,452.040,175.388,14.239,151.996
C06802=1097.404,-107.920,452.049,175.386,14.238,151.996
C06803=1097.399,-108.169,452.060,175.385,14.238,151.997
C06804=1097.392,-108.419,452.070,175.383,14.238,151.997
C06805=1097.386,-108.669,452.079,175.382,14.238,151.997
C06806=1097.380,-108.919,452.089,175.380,14.237,151.998
C06807=1097.374,-109.168,452.099,175.378,14.238,151.998
C06808=1097.368,-109.418,452.108,175.376,14.237,151.999
C06809=1097.361,-109.667,452.118,175.375,14.237,151.999
C06810=1097.355,-109.917,452.128,175.373,14.237,151.999
C06811=1097.349,-110.167,452.137,175.372,14.237,151.999
C06812=1097.344,-110.417,452.148,175.370,14.237,152.000
C06813=1097.337,-110.667,452.157,175.368,14.236,152.000
C06814=1097.331,-110.917,452.167,175.366,14.236,152.001
C06815=1097.325,-111.166,452.176,175.364,14.235,152.001
C06816=1097.319,-111.416,452.186,175.363,14.236,152.001
C06817=1097.312,-111.665,452.196,175.361,14.236,152.002
C06818=1097.306,-111.915,452.206,175.360,14.235,152.002
C06819=1097.301,-112.164,452.215,175.357,14.235,152.002
C06820=1097.294,-112.424,452.225,175.356,14.235,152.003
C06821=1097.288,-112.683,452.235,175.354,14.235,152.003
C06822=1097.281,-112.942,452.245,175.352,14.235,152.003
C06823=1097.275,-113.201,452.255,175.351,14.234,152.004
C06824=1097.269,-113.451,452.265,175.349,14.234,152.004
C06825=1097.263,-113.701,452.275,175.347,14.234,152.004
C06826=1097.257,-113.951,452.284,175.345,14.234,152.005
C06827=1097.251,-114.200,452.294,175.344,14.234,152.005
C06828=1097.245,-114.450,452.303,175.342,14.233,152.005
C06829=1097.239,-114.700,452.313,175.341,14.234,152.006
C06830=1097.232,-114.950,452.322,175.339,14.233,152.006
C06831=1097.226,-115.200,452.332,175.337,14.233,152.006
C06832=1097.220,-115.449,452.342,175.335,14.233,152.007
C06833=1097.214,-115.699,452.351,175.334,14.233,152.007
C06834=1097.208,-115.948,452.360,175.332,14.233,152.008
C06835=1097.202,-116.198,452.370,175.331,14.233,152.008
C06836=1097.196,-116.448,452.380,175.328,14.232,152.008
C06837=1097.190,-116.698,452.389,175.327,14.233,152.009
C06838=1097.184,-116.948,452.399,175.325,14.232,152.009
C06839=1097.177,-117.197,452.408,175.324,14.232,152.009
C06840=1097.171,-117.447,452.418,175.321,14.232,152.010
C06841=1097.164,-117.697,452.427,175.320,14.232,152.010
C06842=1097.158,-117.946,452.436,175.318,14.232,152.010
C06843=1097.152,-118.196,452.446,175.317,14.232,152.011
C06844=1097.146,-118.446,452.455,175.315,14.231,152.011
C06845=1097.140,-118.695,452.465,175.313,14.232,152.011
C06846=1097.134,-118.945,452.474,175.311,14.231,152.012
C06847=1097.128,-119.195,452.484,175.310,14.231,152.012
C06848=1097.122,-119.444,452.493,175.308,14.231,152.013
C06849=1097.116,-119.694,452.503,175.307,14.231,152.013
C06850=1097.109,-119.944,452.512,175.304,14.231,152.013
C06851=1097.104,-120.195,452.521,175.303,14.231,152.014
C06852=1097.097,-120.444,452.531,175.301,14.230,152.014
C06853=1097.090,-120.694,452.540,175.300,14.231,152.014
C06854=1097.084,-120.944,452.549,175.297,14.231,152.015
C06855=1097.079,-121.193,452.559,175.296,14.230,152.015
C06856=1097.073,-121.442,452.568,175.295,14.231,152.015
C06857=1097.066,-121.692,452.578,175.293,14.231,152.016
C06858=1097.060,-121.942,452.587,175.292,14.230,152.016
C06859=1097.054,-122.192,452.597,175.289,14.230,152.016
C06860=1097.048,-122.442,452.606,175.288,14.231,152.017
C06861=1097.041,-122.692,452.615,175.286,14.230,152.017
C06862=1097.035,-122.942,452.624,175.285,14.230,152.017
C06863=1097.029,-123.191,452.634,175.282,14.230,152.018
C06864=1097.023,-123.440,452.643,175.281,14.230,152.018
C06865=1097.017,-123.690,452.653,175.279,14.230,152.019
C06866=1097.011,-123.940,452.662,175.278,14.230,152.019
C06867=1097.005,-124.190,452.671,175.276,14.229,152.019
C06868=1096.998,-124.440,452.680,175.274,14.230,152.020
C06869=1096.992,-124.690,452.690,175.273,14.230,152.020
C06870=1096.986,-124.939,452.699,175.271,14.229,152.020
C06871=1096.980,-125.189,452.708,175.270,14.230,152.021
C06872=1096.974,-125.439,452.717,175.267,14.229,152.021
C06873=1096.968,-125.689,452.726,175.266,14.230,152.022
C06874=1096.961,-125.938,452.736,175.264,14.229,152.022
C06875=1096.955,-126.188,452.745,175.263,14.229,152.022
C06876=1096.949,-126.438,452.755,175.260,14.229,152.023
C06877=1096.943,-126.687,452.763,175.259,14.230,152.023
C06878=1096.937,-126.937,452.772,175.258,14.229,152.023
C06879=1096.931,-127.187,452.782,175.256,14.229,152.024
C06880=1096.924,-127.452,452.792,175.254,14.230,152.024
C06881=1096.917,-127.718,452.801,175.252,14.229,152.025
C06882=1096.911,-127.983,452.811,175.251,14.230,152.025
C06883=1096.907,-128.248,452.822,175.249,14.228,152.025
C06884=1096.499,-128.269,452.714,175.206,14.330,152.054
C06885=1096.501,-128.006,452.703,175.207,14.331,152.054
C06886=1096.508,-127.742,452.694,175.209,14.331,152.054
C06887=1096.514,-127.479,452.684,175.211,14.332,152.054
C06888=1096.521,-127.215,452.675,175.212,14.331,152.053
C06889=1096.527,-126.965,452.665,175.214,14.332,152.053
C06890=1096.533,-126.715,452.656,175.216,14.331,152.052
C06891=1096.539,-126.465,452.646,175.218,14.332,152.052
C06892=1096.545,-126.216,452.638,175.219,14.331,152.052
C06893=1096.551,-125.966,452.629,175.221,14.332,152.051
C06894=1096.558,-125.716,452.619,175.222,14.332,152.051
C06895=1096.564,-125.467,452.609,175.224,14.331,152.051
C06896=1096.570,-125.216,452.601,175.226,14.332,152.050
C06897=1096.577,-124.967,452.592,175.227,14.332,152.050
C06898=1096.583,-124.717,452.582,175.229,14.332,152.050
C06899=1096.588,-124.468,452.573,175.231,14.332,152.049
C06900=1096.594,-124.218,452.563,175.233,14.332,152.049
C06901=1096.601,-123.968,452.554,175.234,14.332,152.048
C06902=1096.607,-123.718,452.545,175.236,14.332,152.048
C06903=1096.613,-123.468,452.536,175.238,14.332,152.048
C06904=1096.620,-123.218,452.526,175.240,14.333,152.047
C06905=1096.625,-122.969,452.517,175.241,14.332,152.047
C06906=1096.631,-122.720,452.508,175.243,14.333,152.047
C06907=1096.638,-122.470,452.499,175.244,14.333,152.046
C06908=1096.644,-122.220,452.490,175.246,14.333,152.046
C06909=1096.650,-121.970,452.480,175.248,14.333,152.046
C06910=1096.656,-121.720,452.471,175.249,14.333,152.045
C06911=1096.663,-121.470,452.461,175.251,14.333,152.045
C06912=1096.669,-121.220,452.451,175.253,14.333,152.045
C06913=1096.674,-120.971,452.442,175.255,14.333,152.044
C06914=1096.681,-120.722,452.433,175.256,14.333,152.044
C06915=1096.687,-120.472,452.423,175.258,14.334,152.043
C06916=1096.694,-120.222,452.414,175.259,14.334,152.043
C06917=1096.699,-119.972,452.405,175.261,14.334,152.043
C06918=1096.706,-119.722,452.396,175.263,14.334,152.042
C06919=1096.712,-119.472,452.386,175.265,14.334,152.042
C06920=1096.718,-119.222,452.377,175.266,14.334,152.042
C06921=1096.724,-118.973,452.367,175.268,14.335,152.042
C06922=1096.730,-118.723,452.357,175.269,14.334,152.041
C06923=1096.736,-118.474,452.348,175.272,14.334,152.041
C06924=1096.742,-118.224,452.339,175.273,14.335,152.040
C06925=1096.748,-117.974,452.329,175.275,14.335,152.040
C06926=1096.754,-117.724,452.320,175.276,14.335,152.040
C06927=1096.761,-117.475,452.310,175.278,14.335,152.039
C06928=1096.767,-117.225,452.300,175.280,14.335,152.039
C06929=1096.774,-116.975,452.291,175.282,14.336,152.039
C06930=1096.780,-116.725,452.282,175.283,14.335,152.038
C06931=1096.786,-116.476,452.272,175.285,14.336,152.038
C06932=1096.792,-116.226,452.263,175.286,14.336,152.038
C06933=1096.798,-115.976,452.253,175.288,14.336,152.037
C06934=1096.805,-115.726,452.244,175.290,14.336,152.037
C06935=1096.810,-115.477,452.234,175.292,14.336,152.037
C06936=1096.816,-115.227,452.225,175.293,14.336,152.036
C06937=1096.822,-114.978,452.215,175.295,14.336,152.036
C06938=1096.829,-114.728,452.206,175.296,14.337,152.036
C06939=1096.835,-114.478,452.196,175.299,14.337,152.035
C06940=1096.841,-114.228,452.187,175.300,14.337,152.035
C06941=1096.847,-113.978,452.177,175.302,14.337,152.035
C06942=1096.853,-113.729,452.167,175.304,14.338,152.034
C06943=1096.859,-113.479,452.158,175.305,14.338,152.034
C06944=1096.865,-113.229,452.148,175.307,14.338,152.034
C06945=1096.872,-112.968,452.138,175.308,14.338,152.033
C06946=1096.878,-112.707,452.128,175.311,14.338,152.033
C06947=1096.884,-112.445,452.118,175.312,14.338,152.033
C06948=1096.891,-112.185,452.108,175.314,14.339,152.032
C06949=1096.897,-111.935,452.098,175.316,14.339,152.032
C06950=1096.903,-111.686,452.088,175.317,14.339,152.031
C06951=1096.910,-111.436,452.079,175.319,14.340,152.031
C06952=1096.915,-111.186,452.069,175.321,14.339,152.031
C06953=1096.921,-110.936,452.059,175.323,14.340,152.031
C06954=1096.927,-110.686,452.050,175.324,14.340,152.030
C06955=1096.934,-110.436,452.040,175.326,14.340,152.030
C06956=1096.940,-110.187,452.030,175.327,14.340,152.029
C06957=1096.946,-109.937,452.020,175.329,14.340,152.029
C06958=1096.952,-109.688,452.011,175.331,14.340,152.029
C06959=1096.958,-109.438,452.001,175.333,14.341,152.028
C06960=1096.965,-109.188,451.991,175.335,14.341,152.028
C06961=1096.971,-108.938,451.982,175.336,14.341,152.028
C06962=1096.977,-108.689,451.971,175.338,14.342,152.027
C06963=1096.983,-108.439,451.961,175.339,14.341,152.027
C06964=1096.989,-108.189,451.952,175.341,14.342,152.027
C06965=1096.995,-107.939,451.942,175.343,14.342,152.026
C06966=1097.001,-107.690,451.933,175.345,14.342,152.026
C06967=1097.007,-107.440,451.923,175.346,14.342,152.026
C06968=1097.014,-107.191,451.913,175.348,14.343,152.025
C06969=1097.019,-106.940,451.903,175.350,14.344,152.025
C06970=1097.026,-106.691,451.893,175.351,14.343,152.025
C06971=1097.032,-106.441,451.884,175.353,14.344,152.025
C06972=1097.038,-106.191,451.874,175.355,14.344,152.024
C06973=1097.044,-105.942,451.864,175.356,14.344,152.024
C06974=1097.050,-105.692,451.854,175.358,14.344,152.023
C06975=1097.056,-105.442,451.844,175.360,14.345,152.023
C06976=1097.062,-105.192,451.834,175.362,14.345,152.023
C06977=1097.069,-104.943,451.824,175.363,14.345,152.023
C06978=1097.074,-104.693,451.814,175.365,14.345,152.022
C06979=1097.080,-104.443,451.804,175.366,14.345,152.022
C06980=1097.086,-104.193,451.795,175.368,14.346,152.022
C06981=1097.093,-103.944,451.785,175.371,14.346,152.021
C06982=1097.098,-103.694,451.774,175.372,14.346,152.021
C06983=1097.104,-103.444,451.765,175.374,14.347,152.021
C06984=1097.111,-103.194,451.755,175.375,14.347,152.020
C06985=1097.117,-102.945,451.745,175.377,14.347,152.020
C06986=1097.123,-102.695,451.735,175.378,14.347,152.020
C06987=1097.129,-102.445,451.725,175.380,14.347,152.019
C06988=1097.135,-102.196,451.715,175.382,14.348,152.019
C06989=1097.141,-101.946,451.705,175.383,14.348,152.019
C06990=1097.147,-101.696,451.695,175.386,14.349,152.018
C06991=1097.153,-101.447,451.685,175.387,14.349,152.018
C06992=1097.159,-101.197,451.675,175.389,14.349,152.018
C06993=1097.165,-100.947,451.665,175.391,14.350,152.017
C06994=1097.171,-100.698,451.655,175.392,14.350,152.017
C06995=1097.178,-100.448,451.645,175.394,14.350,152.017
C06996=1097.183,-100.198,451.635,175.395,14.350,152.016
C06997=1097.189,-99.949,451.625,175.397,14.350,152.016
C06998=1097.196,-99.698,451.615,175.399,14.351,152.016
C06999=1097.202,-99.448,451.605,175.401,14.351,152.015
C07000=1097.208,-99.199,451.595,175.403,14.352,152.015
C07001=1097.214,-98.949,451.585,175.405,14.352,152.015
C07002=1097.221,-98.700,451.575,175.406,14.352,152.014
C07003=1097.226,-98.450,451.565,175.408,14.353,152.014
C07004=1097.232,-98.200,451.555,175.409,14.352,152.014
C07005=1097.239,-97.951,451.545,175.411,14.353,152.013
C07006=1097.244,-97.701,451.535,175.413,14.354,152.013
C07007=1097.251,-97.452,451.524,175.414,14.353,152.013
C07008=1097.256,-97.202,451.514,175.416,14.354,152.013
C07009=1097.263,-96.928,451.503,175.419,14.354,152.012
C07010=1097.269,-96.655,451.492,175.420,14.354,152.012
C07011=1097.276,-96.382,451.480,175.422,14.355,152.011
C07012=1097.283,-96.109,451.470,175.424,14.355,152.011
C07013=1097.289,-95.859,451.460,175.426,14.356,152.011
C07014=1097.294,-95.609,451.449,175.427,14.356,152.011
C07015=1097.301,-95.360,451.440,175.429,14.357,152.010
C07016=1097.306,-95.110,451.429,175.431,14.357,152.010
C07017=1097.313,-94.860,451.419,175.432,14.357,152.010
C07018=1097.319,-94.610,451.408,175.434,14.358,152.009
C07019=1097.325,-94.360,451.399,175.436,14.358,152.009
C07020=1097.331,-94.111,451.388,175.437,14.358,152.009
C07021=1097.337,-93.861,451.378,175.439,14.359,152.008
C07022=1097.343,-93.611,451.367,175.440,14.359,152.008
C07023=1097.349,-93.362,451.358,175.443,14.359,152.008
C07024=1097.355,-93.112,451.347,175.445,14.360,152.007
C07025=1097.360,-92.862,451.337,175.446,14.360,152.007
C07026=1097.367,-92.613,451.326,175.448,14.360,152.007
C07027=1097.372,-92.363,451.316,175.450,14.361,152.007
C07028=1097.379,-92.113,451.306,175.451,14.361,152.006
C07029=1097.384,-91.863,451.295,175.453,14.361,152.006
C07030=1097.391,-91.614,451.285,175.455,14.362,152.006
C07031=1097.397,-91.364,451.274,175.456,14.362,152.005
C07032=1097.403,-91.114,451.265,175.458,14.363,152.005
C07033=1097.409,-90.865,451.254,175.460,14.363,152.005
C07034=1097.415,-90.615,451.244,175.461,14.363,152.004
C07035=1097.421,-90.366,451.233,175.463,14.364,152.004
C07036=1097.427,-90.115,451.223,175.465,14.364,152.004
C07037=1097.433,-89.866,451.213,175.466,14.364,152.004
C07038=1097.439,-89.616,451.202,175.469,14.365,152.003
C07039=1097.445,-89.366,451.192,175.471,14.365,152.003
C07040=1097.451,-89.117,451.181,175.472,14.366,152.003
C07041=1097.457,-88.867,451.172,175.474,14.366,152.002
C07042=1097.463,-88.617,451.160,175.476,14.367,152.002
C07043=1097.470,-88.368,451.150,175.477,14.367,152.002
C07044=1097.475,-88.118,451.140,175.479,14.367,152.001
C07045=1097.481,-87.868,451.129,175.481,14.368,152.001
C07046=1097.487,-87.619,451.119,175.482,14.368,152.001
C07047=1097.493,-87.369,451.109,175.484,14.369,152.001
C07048=1097.500,-87.119,451.098,175.486,14.369,152.000
C07049=1097.506,-86.869,451.087,175.488,14.370,152.000
C07050=1097.511,-86.619,451.077,175.489,14.370,152.000
C07051=1097.517,-86.370,451.067,175.491,14.370,151.999
C07052=1097.523,-86.121,451.056,175.493,14.371,151.999
C07053=1097.530,-85.870,451.046,175.494,14.371,151.999
C07054=1097.536,-85.621,451.035,175.496,14.371,151.998
C07055=1097.541,-85.371,451.024,175.498,14.372,151.998
C07056=1097.548,-85.121,451.015,175.499,14.372,151.998
C07057=1097.553,-84.872,451.004,175.502,14.372,151.997
C07058=1097.560,-84.622,450.993,175.504,14.373,151.997
C07059=1097.566,-84.372,450.982,175.505,14.373,151.997
C07060=1097.572,-84.122,450.972,175.507,14.373,151.996
C07061=1097.578,-83.873,450.962,175.509,14.374,151.996
C07062=1097.584,-83.623,450.950,175.511,14.375,151.996
C07063=1097.590,-83.373,450.940,175.512,14.375,151.996
C07064=1097.596,-83.124,450.930,175.514,14.375,151.995
C07065=1097.602,-82.874,450.919,175.516,14.376,151.995
C07066=1097.609,-82.624,450.908,175.517,14.376,151.995
C07067=1097.615,-82.375,450.898,175.519,14.376,151.994
C07068=1097.620,-82.125,450.887,175.521,14.377,151.994
C07069=1097.627,-81.876,450.877,175.523,14.378,151.994
C07070=1097.633,-81.625,450.866,175.524,14.377,151.993
C07071=1097.639,-81.376,450.855,175.526,14.378,151.993
C07072=1097.645,-81.127,450.845,175.528,14.379,151.993
C07073=1097.652,-80.855,450.833,175.530,14.379,151.992
C07074=1097.658,-80.585,450.822,175.531,14.379,151.992
C07075=1097.665,-80.314,450.810,175.534,14.380,151.992
C07076=1097.671,-80.043,450.798,175.535,14.380,151.991
C07077=1097.678,-79.793,450.788,175.537,14.381,151.991
C07078=1097.684,-79.543,450.777,175.539,14.382,151.991
C07079=1097.689,-79.293,450.766,175.541,14.381,151.991
C07080=1097.695,-79.044,450.756,175.543,14.382,151.990
C07081=1097.701,-78.794,450.744,175.544,14.383,151.990
C07082=1097.708,-78.544,450.734,175.546,14.384,151.990
C07083=1097.714,-78.295,450.723,175.548,14.383,151.989
C07084=1097.719,-78.045,450.712,175.550,14.384,151.989
C07085=1097.726,-77.795,450.701,175.551,14.385,151.989
C07086=1097.731,-77.545,450.691,175.553,14.386,151.989
C07087=1097.737,-77.296,450.680,175.555,14.385,151.988
C07088=1097.743,-77.046,450.670,175.557,14.386,151.988
C07089=1097.750,-76.796,450.659,175.559,14.387,151.988
C07090=1097.755,-76.547,450.648,175.560,14.387,151.987
C07091=1097.761,-76.297,450.637,175.562,14.388,151.987
C07092=1097.767,-76.047,450.626,175.564,14.388,151.987
C07093=1097.773,-75.798,450.615,175.566,14.389,151.986
C07094=1097.779,-75.548,450.604,175.567,14.389,151.986
C07095=1097.785,-75.299,450.593,175.569,14.389,151.986
C07096=1097.792,-75.049,450.582,175.571,14.390,151.985
C07097=1097.798,-74.799,450.571,175.573,14.390,151.985
C07098=1097.803,-74.550,450.560,175.575,14.391,151.985
C07099=1097.810,-74.299,450.549,175.576,14.391,151.985
C07100=1097.815,-74.050,450.538,175.578,14.392,151.984
C07101=1097.821,-73.801,450.527,175.580,14.392,151.984
C07102=1097.827,-73.550,450.517,175.582,14.393,151.984
C07103=1097.833,-73.300,450.506,175.583,14.394,151.983
C07104=1097.839,-73.051,450.495,175.585,14.394,151.983
C07105=1097.844,-72.801,450.484,175.586,14.395,151.983
C07106=1097.850,-72.552,450.473,175.589,14.395,151.983
C07107=1097.856,-72.302,450.462,175.591,14.396,151.982
C07108=1097.862,-72.052,450.451,175.592,14.396,151.982
C07109=1097.868,-71.803,450.440,175.594,14.397,151.982
C07110=1097.874,-71.553,450.430,175.595,14.397,151.982
C07111=1097.880,-71.304,450.418,175.597,14.398,151.981
C07112=1097.886,-71.054,450.407,175.599,14.399,151.981
C07113=1097.892,-70.805,450.396,175.601,14.398,151.981
C07114=1097.898,-70.554,450.385,175.602,14.399,151.980
C07115=1097.904,-70.305,450.374,175.604,14.400,151.980
C07116=1097.909,-70.055,450.362,175.606,14.401,151.980
C07117=1097.915,-69.805,450.351,175.608,14.401,151.980
C07118=1097.921,-69.555,450.340,175.609,14.402,151.979
C07119=1097.927,-69.306,450.329,175.611,14.402,151.979
C07120=1097.932,-69.056,450.318,175.613,14.403,151.979
C07121=1097.939,-68.806,450.307,175.615,14.403,151.978
C07122=1097.944,-68.557,450.296,175.617,14.404,151.978
C07123=1097.950,-68.307,450.285,175.618,14.404,151.978
C07124=1097.957,-68.058,450.273,175.620,14.405,151.978
C07125=1097.963,-67.808,450.263,175.622,14.405,151.977
C07126=1097.968,-67.559,450.252,175.624,14.406,151.977
C07127=1097.974,-67.308,450.240,175.626,14.407,151.977
C07128=1097.980,-67.059,450.229,175.627,14.407,151.976
C07129=1097.985,-66.809,450.218,175.629,14.408,151.976
C07130=1097.992,-66.559,450.207,175.631,14.408,151.976
C07131=1097.998,-66.310,450.195,175.633,14.409,151.975
C07132=1098.004,-66.060,450.184,175.635,14.409,151.975
C07133=1098.010,-65.810,450.173,175.636,14.409,151.975
C07134=1098.016,-65.561,450.162,175.638,14.410,151.975
C07135=1098.022,-65.311,450.151,175.640,14.411,151.974
C07136=1098.027,-65.061,450.140,175.642,14.412,151.974
C07137=1098.034,-64.792,450.127,175.644,14.412,151.974
C07138=1098.040,-64.524,450.116,175.646,14.413,151.974
C07139=1098.046,-64.254,450.103,175.648,14.413,151.973
C07140=1098.053,-63.986,450.091,175.650,14.414,151.973
C07141=1098.059,-63.737,450.079,175.652,14.414,151.973
C07142=1098.065,-63.487,450.069,175.653,14.415,151.972
C07143=1098.071,-63.238,450.058,175.655,14.415,151.972
C07144=1098.076,-62.987,450.046,175.657,14.416,151.972
C07145=1098.082,-62.738,450.034,175.658,14.417,151.972
C07146=1098.089,-62.488,450.023,175.661,14.417,151.971
C07147=1098.095,-62.239,450.012,175.663,14.418,151.971
C07148=1098.101,-61.988,450.001,175.664,14.418,151.971
C07149=1098.107,-61.740,449.989,175.665,14.419,151.970
C07150=1098.112,-61.490,449.978,175.667,14.419,151.970
C07151=1098.118,-61.240,449.967,175.669,14.420,151.970
C07152=1098.124,-60.991,449.955,175.671,14.420,151.969
C07153=1098.131,-60.741,449.944,175.673,14.421,151.969
C07154=1098.136,-60.491,449.933,175.675,14.422,151.969
C07155=1098.142,-60.241,449.920,175.676,14.422,151.969
C07156=1098.148,-59.992,449.909,175.678,14.423,151.968
C07157=1098.154,-59.741,449.898,175.680,14.423,151.968
C07158=1098.160,-59.493,449.887,175.682,14.424,151.968
C07159=1098.167,-59.242,449.875,175.684,14.425,151.967
C07160=1098.172,-58.993,449.864,175.686,14.425,151.967
C07161=1098.178,-58.744,449.852,175.687,14.425,151.967
C07162=1098.184,-58.494,449.841,175.689,14.426,151.967
C07163=1098.190,-58.244,449.830,175.691,14.426,151.966
C07164=1098.197,-57.994,449.818,175.693,14.427,151.966
C07165=1098.202,-57.745,449.807,175.695,14.428,151.966
C07166=1098.208,-57.495,449.795,175.697,14.429,151.965
C07167=1098.214,-57.246,449.784,175.699,14.429,151.965
C07168=1098.220,-56.995,449.773,175.700,14.429,151.965
C07169=1098.226,-56.746,449.760,175.702,14.430,151.965
C07170=1098.232,-56.496,449.749,175.704,14.431,151.964
C07171=1098.239,-56.246,449.737,175.706,14.431,151.964
C07172=1098.244,-55.997,449.726,175.708,14.432,151.964
C07173=1098.250,-55.747,449.714,175.710,14.432,151.963
C07174=1098.256,-55.498,449.703,175.712,14.433,151.963
C07175=1098.263,-55.248,449.691,175.714,14.434,151.963
C07176=1098.268,-54.999,449.680,175.715,14.434,151.963
C07177=1098.274,-54.749,449.668,175.717,14.435,151.962
C07178=1098.280,-54.499,449.657,175.719,14.435,151.962
C07179=1098.286,-54.249,449.645,175.721,14.436,151.962
C07180=1098.292,-54.000,449.634,175.723,14.436,151.961
C07181=1098.298,-53.750,449.622,175.724,14.437,151.961
C07182=1098.304,-53.501,449.610,175.726,14.438,151.961
C07183=1098.311,-53.251,449.598,175.728,14.438,151.960
C07184=1098.316,-53.001,449.587,175.730,14.438,151.960
C07185=1098.322,-52.752,449.575,175.731,14.439,151.960
C07186=1098.329,-52.502,449.564,175.733,14.440,151.960
C07187=1098.335,-52.253,449.552,175.735,14.441,151.959
C07188=1098.340,-52.002,449.540,175.737,14.441,151.959
C07189=1098.347,-51.753,449.528,175.739,14.442,151.959
C07190=1098.353,-51.503,449.517,175.741,14.442,151.958
C07191=1098.359,-51.253,449.505,175.743,14.443,151.958
C07192=1098.365,-51.004,449.493,175.745,14.444,151.958
C07193=1098.371,-50.754,449.482,175.746,14.444,151.957
C07194=1098.377,-50.504,449.470,175.748,14.444,151.957
C07195=1098.383,-50.255,449.459,175.750,14.445,151.957
C07196=1098.389,-50.005,449.446,175.752,14.446,151.957
C07197=1098.394,-49.755,449.435,175.754,14.447,151.956
C07198=1098.400,-49.506,449.423,175.756,14.447,151.956
C07199=1098.406,-49.257,449.411,175.758,14.448,151.956
C07200=1098.412,-49.006,449.399,175.760,14.448,151.955
C07201=1098.418,-48.739,449.387,175.762,14.449,151.955
C07202=1098.425,-48.472,449.374,175.764,14.450,151.955
C07203=1098.431,-48.204,449.361,175.765,14.451,151.955
C07204=1098.437,-47.937,449.349,175.767,14.451,151.954
C07205=1098.443,-47.688,449.336,175.769,14.452,151.954
C07206=1098.449,-47.437,449.325,175.771,14.452,151.954
C07207=1098.454,-47.188,449.313,175.773,14.453,151.953
C07208=1098.461,-46.939,449.301,175.775,14.454,151.953
C07209=1098.466,-46.688,449.289,175.777,14.455,151.953
C07210=1098.472,-46.439,449.278,175.779,14.455,151.953
C07211=1098.478,-46.189,449.265,175.780,14.456,151.952
C07212=1098.483,-45.940,449.254,175.782,14.456,151.952
C07213=1098.490,-45.690,449.242,175.784,14.457,151.952
C07214=1098.496,-45.440,449.229,175.786,14.457,151.952
C07215=1098.502,-45.191,449.217,175.788,14.458,151.951
C07216=1098.508,-44.941,449.206,175.790,14.459,151.951
C07217=1098.514,-44.692,449.194,175.792,14.460,151.951
C07218=1098.520,-44.442,449.181,175.793,14.460,151.950
C07219=1098.525,-44.191,449.170,175.795,14.461,151.950
C07220=1098.531,-43.943,449.158,175.798,14.461,151.950
C07221=1098.537,-43.693,449.145,175.799,14.462,151.950
C07222=1098.543,-43.444,449.134,175.801,14.463,151.949
C07223=1098.549,-43.194,449.121,175.803,14.464,151.949
C07224=1098.555,-42.943,449.109,175.805,14.464,151.949
C07225=1098.561,-42.695,449.098,175.807,14.465,151.948
C07226=1098.567,-42.445,449.085,175.808,14.465,151.948
C07227=1098.573,-42.195,449.073,175.810,14.465,151.948
C07228=1098.579,-41.946,449.061,175.812,14.466,151.948
C07229=1098.584,-41.695,449.049,175.814,14.467,151.947
C07230=1098.591,-41.446,449.037,175.816,14.468,151.947
C07231=1098.596,-41.197,449.025,175.818,14.469,151.947
C07232=1098.602,-40.947,449.013,175.820,14.469,151.946
C07233=1098.609,-40.697,449.001,175.822,14.470,151.946
C07234=1098.614,-40.448,448.988,175.824,14.470,151.946
C07235=1098.620,-40.198,448.977,175.826,14.471,151.946
C07236=1098.626,-39.948,448.965,175.827,14.472,151.945
C07237=1098.632,-39.699,448.953,175.829,14.473,151.945
C07238=1098.638,-39.449,448.941,175.831,14.473,151.945
C07239=1098.644,-39.199,448.928,175.833,14.474,151.944
C07240=1098.649,-38.950,448.916,175.835,14.474,151.944
C07241=1098.655,-38.700,448.903,175.837,14.475,151.944
C07242=1098.662,-38.451,448.891,175.839,14.476,151.944
